	#AI_2(i_iRawSignal := 27648,
	      io_stConfig := "DB_Test_IO".Config[2],
	      io_stOut := "DB_Test_IO".Out[2]);
	#Alarm_2(i_rValue := "DB_Test_IO".Out[2].Value_Filtered, i_boReset := "DB_Test_IO".Reset_Alarms, i_boInhibit := False, io_stConfig := "DB_Test_IO".Alarm_Cfg[2], io_stOut := "DB_Test_IO".Alarm_Out[2]);
	
END_FUNCTION_BLOCK

FUNCTION_BLOCK "FB_Sim_SawTooth_UpDown"
{ S7_Optimized_Access := 'FALSE' }
VERSION : 0.1
   VAR_INPUT 
      Enable : Bool;
      Speed : Real;
      Limit_High : Int := 27648;   // Верхний предел (по умолчанию максимум для аналогового входа Siemens)
      Limit_Low : Int := 0;   // Нижний предел
   END_VAR

   VAR_OUTPUT 
      Out_Raw : Int;
   END_VAR

   VAR_IN_OUT 
      Current_Val : Int;
   END_VAR

   VAR 
      Dir_Up : Bool := TRUE;   // Направление: TRUE = вверх, FALSE = вниз
   END_VAR

   VAR_TEMP 
      Increment : Int;
   END_VAR


BEGIN
	    // Если блок выключен, замораживаем текущее значение, сохраняем направление и выходим
	    IF NOT #Enable THEN
	        #Out_Raw := #Current_Val;
	        RETURN;
	    END_IF;
	    
	    // Рассчитываем шаг за цикл
	    #Increment := REAL_TO_INT(ABS(#Speed) * "getCycleTime"() / 1000.0);
	    
	    // Логика треугольного сигнала ("вверх-вниз")
	    IF #Dir_Up THEN
	        // Считаем вверх
	        #Current_Val := #Current_Val + #Increment;
	        IF #Current_Val >= #Limit_High THEN
	            #Current_Val := #Limit_High;
	            #Dir_Up := FALSE; // Меняем направление на "вниз"
	        END_IF;
	    ELSE
	        // Считаем вниз
	        #Current_Val := #Current_Val - #Increment;
	        IF #Current_Val <= #Limit_Low THEN
	            #Current_Val := #Limit_Low;
	            #Dir_Up := TRUE;  // Меняем направление на "вверх"
	        END_IF;
	    END_IF;
	    
	    // Обновляем выход
	    #Out_Raw := #Current_Val;
	    
END_FUNCTION_BLOCK

FUNCTION "getCycleTime" : Real
{ S7_Optimized_Access := 'FALSE' }
VERSION : 0.1

BEGIN
	#getCycleTime := "DB_Global".Sys.CycleTime_ms_REAL;
END_FUNCTION

FUNCTION_BLOCK "FB_RawDistort"
{ S7_Optimized_Access := 'FALSE' }
VERSION : 0.1
// 5. BLOCKS (FB_RawDistort, FB_Sim_SawTooth, FB_AI, FB_AnalogAlarm)
   VAR_INPUT 
      Enable : Bool;
      RawIn : Int;
      Dt_ms : Real;
      NoiseAmpRaw : Int;
      Noise_Hz : Real;
      StepTrig : Bool;
      StepRaw : Int;
      StepHold_ms : DInt;
   END_VAR

   VAR_OUTPUT 
      RawOut : Int;
   END_VAR

   VAR 
      phase : Real;
      noiseVal : Real;
      step_active : Bool;
      step_left_ms : DInt;
      step_prev : Bool;
   END_VAR


BEGIN
	
	IF NOT #Enable THEN
	    #RawOut := #RawIn;
	    RETURN;
	END_IF;
	#phase := #phase + (6.283185 * #Noise_Hz * #Dt_ms * 0.001);
	IF #phase > 6.283185 THEN
	    #phase := #phase - 6.283185;
	END_IF;
	#noiseVal := SIN(#phase);
	IF (#StepTrig AND NOT #step_prev) THEN
	    #step_active := TRUE;
	    #step_left_ms := #StepHold_ms;
	END_IF;
	#step_prev := #StepTrig;
	IF #step_active THEN
	    IF #step_left_ms > REAL_TO_DINT(#Dt_ms) THEN
	        #step_left_ms := #step_left_ms - REAL_TO_DINT(#Dt_ms);
	    ELSE
	        #step_active := FALSE;
	    END_IF;
	END_IF;
	#RawOut := REAL_TO_INT(INT_TO_REAL(#RawIn) + (#noiseVal * INT_TO_REAL(#NoiseAmpRaw)));
	
END_FUNCTION_BLOCK

FUNCTION_BLOCK "FB_AI"
{ S7_Optimized_Access := 'FALSE' }
VERSION : 7.9
// -----------------------------------------------------------------------------
// БЛОК ОБРАБОТКИ АНАЛОГОВОГО СИГНАЛА (FB_AI)
// -----------------------------------------------------------------------------
   VAR_INPUT 
      i_iRawSignal : Int;
      i_rSimValue : Real;
   END_VAR

   VAR_IN_OUT 
      io_stConfig : "UDT_AI_Config";
      io_stOut : "UDT_AI_Out";
   END_VAR

   VAR 
      stat_boWasInvalid : Bool := TRUE;
   END_VAR

   VAR_TEMP 
      temp_boDisabled : Bool;
      temp_boSimActive : Bool;
      temp_boUseSqrt : Bool;
      temp_boPreSqrtCut : Bool;
      temp_boFinalClamp : Bool;
      temp_rMA : Real;
      temp_rNorm : Real;
      temp_rCutoff_Norm : Real;
      temp_rScaled : Real;
      temp_rRange_mA : Real;
      temp_rRange_Phys : Real;
      temp_rMinPhys : Real;
      temp_rMaxPhys : Real;
      temp_boResetFilter : Bool;
      temp_iFilterTime : Int;
   END_VAR


BEGIN
	    // =========================================================
	    // ШАГ 0. РАСШИФРОВКА БИТОВОГО СЛОВА (Mode)
	    // =========================================================
	    #temp_boDisabled := (#io_stConfig.Mode AND 16#0001) = 16#0001;
	    #temp_boSimActive := (#io_stConfig.Mode AND 16#0002) = 16#0002;
	    #temp_boUseSqrt := (#io_stConfig.Mode AND 16#0004) = 16#0004;
	    #temp_boPreSqrtCut := (#io_stConfig.Mode AND 16#0008) = 16#0008;
	    #temp_boFinalClamp := (#io_stConfig.Mode AND 16#0010) = 16#0010;
	    
	    // 0.1 Режим полного отключения канала
	    IF #temp_boDisabled THEN
	        #io_stOut.Value_Unclamped := 0.0;
	        #io_stOut.Value_Scaled := 0.0;
	        #io_stOut.Value_Filtered := 0.0;
	        #io_stOut.Value_mA := 0.0;
	        #io_stOut.Raw := 0;
	        
	        #io_stOut.Status.WireBreak := FALSE;
	        #io_stOut.Status.Underrange := FALSE;
	        #io_stOut.Status.Overrange := FALSE;
	        #io_stOut.Status.Overflow := FALSE;
	        #io_stOut.Status.ConfigError := FALSE;
	        #io_stOut.Status.Sim_Active := FALSE;
	        
	        #stat_boWasInvalid := TRUE;
	        RETURN;
	    END_IF;
	    
	    // 0.2 Защита от кривых настроек
	    #temp_rRange_mA := #io_stConfig.Calib_mA_Max - #io_stConfig.Calib_mA_Min;
	    #temp_rRange_Phys := #io_stConfig.Scale_Max - #io_stConfig.Scale_Min;
	    
	    IF (#io_stConfig.HW_Max <= #io_stConfig.HW_Min) OR
	        (#temp_rRange_mA <= 0.0) OR
	        (ABS(#temp_rRange_Phys) < 0.00001) OR
	        (ABS(#io_stConfig.Cutoff) >= ABS(#temp_rRange_Phys)) THEN
	        
	        #io_stOut.Status.ConfigError := TRUE;
	        
	        #io_stOut.Status.WireBreak := FALSE;
	        #io_stOut.Status.Underrange := FALSE;
	        #io_stOut.Status.Overrange := FALSE;
	        #io_stOut.Status.Overflow := FALSE;
	        #io_stOut.Status.Sim_Active := FALSE;
	        
	        #io_stOut.Value_Unclamped := 0.0;
	        #io_stOut.Value_Scaled := 0.0;
	        #io_stOut.Value_Filtered := 0.0;
	        #io_stOut.Value_mA := 0.0;
	        #io_stOut.Raw := #i_iRawSignal;
	        
	        #stat_boWasInvalid := TRUE;
	        RETURN;
	    END_IF;
	    
	    #io_stOut.Status.ConfigError := FALSE;
	    
	    // =========================================================
	    // ШАГ 1 & 2. СИМУЛЯЦИЯ И ДИАГНОСТИКА
	    // =========================================================
	    
	    IF #temp_boSimActive THEN
	        #io_stOut.Status.Sim_Active := TRUE;
	        
	        #io_stOut.Status.WireBreak := FALSE;
	        #io_stOut.Status.Underrange := FALSE;
	        #io_stOut.Status.Overrange := FALSE;
	        #io_stOut.Status.Overflow := FALSE;
	        
	        #io_stOut.Raw := 0;
	        #io_stOut.Value_mA := 0.0;
	        #temp_rScaled := #i_rSimValue;
	    ELSE
	        #io_stOut.Status.Sim_Active := FALSE;
	        #io_stOut.Raw := #i_iRawSignal;
	        
	        "FC_AnalogDiag"(
	                        i_iRawSignal := #i_iRawSignal,
	                        i_iHW_Min := #io_stConfig.HW_Min,
	                        i_iHW_Max := #io_stConfig.HW_Max,
	                        i_rCoef_Under := "C_DIAG_UNDER",
	                        i_rCoef_Over := "C_DIAG_OVER",
	                        o_boWireBreak => #io_stOut.Status.WireBreak,
	                        o_boUnderrange => #io_stOut.Status.Underrange,
	                        o_boOverrange => #io_stOut.Status.Overrange,
	                        o_boOverflow => #io_stOut.Status.Overflow
	        );
	        
	        // =========================================================
	        // ШАГ 3. МАТЕМАТИКА
	        // =========================================================
	        IF #io_stOut.Status.WireBreak THEN
	            // Ушли в жесткий минус: База + (Диапазон * Коэффициент обрыва)
	            #temp_rScaled := #io_stConfig.Scale_Min + (#temp_rRange_Phys * "C_DIAG_UNDER");
	            #io_stOut.Value_mA := 0.0;
	            
	        ELSIF #io_stOut.Status.Overflow THEN
	            // Ушли в жесткий перегруз: База + (Диапазон * Коэффициент переполнения)
	            #temp_rScaled := #io_stConfig.Scale_Min + (#temp_rRange_Phys * "C_DIAG_OVER");
	            #io_stOut.Value_mA := 25.0;
	        ELSE
	            // А) Расчет миллиампер
	            #temp_rMA := 4.0 + ((INT_TO_REAL(#i_iRawSignal) - INT_TO_REAL(#io_stConfig.HW_Min)) /
	            (INT_TO_REAL(#io_stConfig.HW_Max) - INT_TO_REAL(#io_stConfig.HW_Min))) * 16.0;
	            #io_stOut.Value_mA := #temp_rMA;
	            
	            // Б) Нормализация (0.0 ... 1.0)
	            #temp_rNorm := (#temp_rMA - #io_stConfig.Calib_mA_Min) / #temp_rRange_mA;
	            
	            // В) Pre-Sqrt CutOff (Умная отсечка до извлечения корня)
	            IF #temp_boPreSqrtCut AND #temp_boUseSqrt THEN
	                #temp_rCutoff_Norm := ABS(#io_stConfig.Cutoff / #temp_rRange_Phys);
	                #temp_rCutoff_Norm := #temp_rCutoff_Norm * #temp_rCutoff_Norm;
	                
	                IF #temp_rNorm < #temp_rCutoff_Norm THEN
	                    #temp_rNorm := 0.0;
	                END_IF;
	            END_IF;
	            
	            // Г) Извлечение корня
	            IF #temp_boUseSqrt THEN
	                IF #temp_rNorm > 0.0 THEN
	                    #temp_rNorm := SQRT(#temp_rNorm);
	                ELSE
	                    #temp_rNorm := 0.0;
	                END_IF;
	            END_IF;
	            
	            // Д) Масштабирование в физическую величину
	            #temp_rScaled := #io_stConfig.Scale_Min + (#temp_rNorm * #temp_rRange_Phys);
	            
	            // Е) Классический CutOff 
	            IF NOT (#temp_boPreSqrtCut AND #temp_boUseSqrt) THEN
	                IF ABS(#temp_rScaled) < ABS(#io_stConfig.Cutoff) THEN
	                    #temp_rScaled := 0.0;
	                END_IF;
	            END_IF;
	        END_IF;
	    END_IF;
	    
	    // Сохраняем чистую математику (без клампа) на выход
	    #io_stOut.Value_Unclamped := #temp_rScaled;
	    
	    // =========================================================
	    // ШАГ 3.5. ФИНАЛЬНЫЙ CLAMP (Beautiful Branch)
	    // =========================================================
	    IF #temp_boFinalClamp THEN
	        #temp_rMinPhys := MIN(IN1 := #io_stConfig.Scale_Min, IN2 := #io_stConfig.Scale_Max);
	        #temp_rMaxPhys := MAX(IN1 := #io_stConfig.Scale_Min, IN2 := #io_stConfig.Scale_Max);
	        #temp_rScaled := LIMIT(MN := #temp_rMinPhys, IN := #temp_rScaled, MX := #temp_rMaxPhys);
	    END_IF;
	    
	    #io_stOut.Value_Scaled := #temp_rScaled;
	    
	    // =========================================================
	    // ШАГ 4. ФИЛЬТРАЦИЯ & PRE-LOAD 
	    // =========================================================
	    #temp_boResetFilter := #temp_boSimActive OR
	    #io_stOut.Status.WireBreak OR
	    #io_stOut.Status.Overflow OR
	    #stat_boWasInvalid;
	    
	    #temp_iFilterTime := LIMIT(MN := 0, IN := #io_stConfig.FilterTime_ms, MX := 32000);
	    
	    "FC_Filter_PT1"(
	                    i_rRawValue := #temp_rScaled, // Фильтруем заклампованное значение
	                    i_rTimeFilter_ms := INT_TO_REAL(#temp_iFilterTime),
	                    i_boReset := #temp_boResetFilter,
	                    io_rFilteredValue := #io_stOut.Value_Filtered
	    );
	    
	    #stat_boWasInvalid := #io_stOut.Status.WireBreak OR
	    #io_stOut.Status.Overflow OR
	    #io_stOut.Status.ConfigError;
	    
END_FUNCTION_BLOCK

FUNCTION "FC_AnalogDiag" : Void
{ S7_Optimized_Access := 'FALSE' }
VERSION : 1.1
   VAR_INPUT 
      i_iRawSignal : Int;
      i_iHW_Min : Int;
      i_iHW_Max : Int;
      i_rCoef_Under : Real;
      i_rCoef_Over : Real;
   END_VAR

   VAR_OUTPUT 
      o_boWireBreak : Bool;
      o_boUnderrange : Bool;
      o_boOverrange : Bool;
      o_boOverflow : Bool;
   END_VAR

   VAR_TEMP 
      temp_rLimit_Max : Real;
      temp_iLimit_Min : Int;
   END_VAR


BEGIN
	    #temp_rLimit_Max := INT_TO_REAL(#i_iHW_Max) * #i_rCoef_Over;
	    #temp_iLimit_Min := REAL_TO_INT(INT_TO_REAL(#i_iHW_Max) * #i_rCoef_Under);
	    
	    #o_boWireBreak := #i_iRawSignal < #temp_iLimit_Min;
	    #o_boUnderrange := (#i_iRawSignal < #i_iHW_Min) AND (#i_iRawSignal >= #temp_iLimit_Min);
	    #o_boOverrange := (#i_iRawSignal > #i_iHW_Max) AND (#i_iRawSignal <= REAL_TO_INT(#temp_rLimit_Max));
	    #o_boOverflow := #i_iRawSignal > REAL_TO_INT(#temp_rLimit_Max);
END_FUNCTION

FUNCTION "FC_Filter_PT1" : Void
{ S7_Optimized_Access := 'FALSE' }
VERSION : 0.1
   VAR_INPUT 
      i_rRawValue : Real;
      i_rTimeFilter_ms : Real;
      i_boReset : Bool;
   END_VAR

   VAR_IN_OUT 
      io_rFilteredValue : Real;
   END_VAR

   VAR_TEMP 
      temp_rCycleTime_ms : Real;
      temp_rAlpha : Real;
   END_VAR


BEGIN
	
	IF #i_boReset THEN
	    #io_rFilteredValue := #i_rRawValue;
	    RETURN;
	END_IF;
	#temp_rCycleTime_ms := "getCycleTime"();
	IF #temp_rCycleTime_ms <= 0.000001 THEN
	    RETURN;
	END_IF;
	#temp_rAlpha := #temp_rCycleTime_ms / (#i_rTimeFilter_ms + #temp_rCycleTime_ms);
	#io_rFilteredValue := #io_rFilteredValue + #temp_rAlpha * (#i_rRawValue - #io_rFilteredValue);
	
	
	
END_FUNCTION

FUNCTION_BLOCK "FB_AnalogAlarm"
{ S7_Optimized_Access := 'FALSE' }
VERSION : 2.0
   VAR_INPUT 
      i_rValue : Real;
      i_boReset : Bool;
      i_boInhibit : Bool;
   END_VAR

   VAR_IN_OUT 
      io_stConfig : "UDT_Alarm_Config";
      io_stOut : "UDT_Alarm_Out";
   END_VAR

   VAR 
      stat_TonHiHi {InstructionName := 'TON'; LibVersion := '1.0'; S7_SetPoint := 'False'} : TON;
      stat_TonHi {InstructionName := 'TON'; LibVersion := '1.0'; S7_SetPoint := 'False'} : TON;
      stat_TonLo {InstructionName := 'TON'; LibVersion := '1.0'; S7_SetPoint := 'False'} : TON;
      stat_TonLoLo {InstructionName := 'TON'; LibVersion := '1.0'; S7_SetPoint := 'False'} : TON;
      stat_RawHiHi : Bool;
      stat_RawHi : Bool;
      stat_RawLo : Bool;
      stat_RawLoLo : Bool;
   END_VAR


BEGIN
	    // =========================================================
	    // 1. ТРАНСЛЯЦИЯ СТАТУСОВ ДЛЯ HMI (En_Out)
	    // =========================================================
	    #io_stOut.En_HiHi := #io_stConfig.En_Alarm.HiHi AND NOT #i_boInhibit ;
	    #io_stOut.En_Hi := #io_stConfig.En_Alarm.Hi AND NOT #i_boInhibit;
	    #io_stOut.En_Lo := #io_stConfig.En_Alarm.Lo AND NOT #i_boInhibit;
	    #io_stOut.En_LoLo := #io_stConfig.En_Alarm.LoLo AND NOT #i_boInhibit;
	    #io_stOut.En_Latch_Enable := #io_stConfig.En_Alarm.Latch_Enable;
	    
	    // =========================================================
	    // 2. ОБРАБОТКА СЫРЫХ АВАРИЙ С ГИСТЕРЕЗИСОМ (Deadband)
	    // =========================================================
	    // Верхние пороги (Срабатывание >, Сброс <)
	    IF #i_rValue > #io_stConfig.HiHi THEN
	        #stat_RawHiHi := TRUE;
	    ELSIF #i_rValue < (#io_stConfig.HiHi - #io_stConfig.Hysteresis) THEN
	        #stat_RawHiHi := FALSE;
	    END_IF;
	    
	    IF #i_rValue > #io_stConfig.Hi THEN
	        #stat_RawHi := TRUE;
	    ELSIF #i_rValue < (#io_stConfig.Hi - #io_stConfig.Hysteresis) THEN
	        #stat_RawHi := FALSE;
	    END_IF;
	    
	    // Нижние пороги (Срабатывание <, Сброс >)
	    IF #i_rValue < #io_stConfig.Lo THEN
	        #stat_RawLo := TRUE;
	    ELSIF #i_rValue > (#io_stConfig.Lo + #io_stConfig.Hysteresis) THEN
	        #stat_RawLo := FALSE;
	    END_IF;
	    
	    IF #i_rValue < #io_stConfig.LoLo THEN
	        #stat_RawLoLo := TRUE;
	    ELSIF #i_rValue > (#io_stConfig.LoLo + #io_stConfig.Hysteresis) THEN
	        #stat_RawLoLo := FALSE;
	    END_IF;
	    
	    // =========================================================
	    // 3. ТАЙМЕРЫ ЗАДЕРЖКИ (ON-Delay)
	    // =========================================================
	    // Таймер не считает, если сработала блокировка датчика (Inhibit) 
	    // или аларм выключен в настройках.
	    #stat_TonHiHi(IN := #stat_RawHiHi AND #io_stConfig.En_Alarm.HiHi AND NOT #i_boInhibit,
	                  PT := DINT_TO_TIME(#io_stConfig.Delay_HiHi)*1000 );
	    
	    #stat_TonHi(IN := #stat_RawHi AND #io_stConfig.En_Alarm.Hi AND NOT #i_boInhibit,
	                PT := DINT_TO_TIME(#io_stConfig.Delay_Hi)*1000 );
	    
	    #stat_TonLo(IN := #stat_RawLo AND #io_stConfig.En_Alarm.Lo AND NOT #i_boInhibit,
	                PT := DINT_TO_TIME(#io_stConfig.Delay_Lo)*1000 );
	    
	    #stat_TonLoLo(IN := #stat_RawLoLo AND #io_stConfig.En_Alarm.LoLo AND NOT #i_boInhibit,
	                  PT := DINT_TO_TIME(#io_stConfig.Delay_LoLo)*1000 );
	    
	    // =========================================================
	    // 4. ФИКСАЦИЯ (LATCH) И СБРОС АВАРИЙ
	    // =========================================================
	    // Логика сброса (имеет приоритет):
	    // 1. Сработал Inhibit (глушим всё безусловно)
	    // 2. Аларм сняли в настройках
	    // 3. Уровень в норме И (нет фиксации ИЛИ нажата кнопка Reset)
	    
	    // --- HiHi ---
	    IF #i_boInhibit OR NOT #io_stConfig.En_Alarm.HiHi OR
	        (NOT #stat_RawHiHi AND (NOT #io_stConfig.En_Alarm.Latch_Enable OR #i_boReset)) THEN
	        #io_stOut.HiHi := FALSE;
	    ELSIF #stat_TonHiHi.Q THEN
	        #io_stOut.HiHi := TRUE;
	    END_IF;
	    
	    // --- Hi ---
	    IF #i_boInhibit OR NOT #io_stConfig.En_Alarm.Hi OR
	        (NOT #stat_RawHi AND (NOT #io_stConfig.En_Alarm.Latch_Enable OR #i_boReset)) THEN
	        #io_stOut.Hi := FALSE;
	    ELSIF #stat_TonHi.Q THEN
	        #io_stOut.Hi := TRUE;
	    END_IF;
	    
	    // --- Lo ---
	    IF #i_boInhibit OR NOT #io_stConfig.En_Alarm.Lo OR
	        (NOT #stat_RawLo AND (NOT #io_stConfig.En_Alarm.Latch_Enable OR #i_boReset)) THEN
	        #io_stOut.Lo := FALSE;
	    ELSIF #stat_TonLo.Q THEN
	        #io_stOut.Lo := TRUE;
	    END_IF;
	    
	    // --- LoLo ---
	    IF #i_boInhibit OR NOT #io_stConfig.En_Alarm.LoLo OR
	        (NOT #stat_RawLoLo AND (NOT #io_stConfig.En_Alarm.Latch_Enable OR #i_boReset)) THEN
	        #io_stOut.LoLo := FALSE;
	    ELSIF #stat_TonLoLo.Q THEN
	        #io_stOut.LoLo := TRUE;
	    END_IF;
	    
END_FUNCTION_BLOCK

FUNCTION "FC_Wh_TRN_Mng" : Void
{ S7_Optimized_Access := 'FALSE' }
VERSION : 0.1
   VAR_TEMP 
      temp_Ind : Int;
   END_VAR


BEGIN
	// ---------------------------------------------------------------
	// Склад: Транзитный (TRN) — 2 весовых и 1 аналоговый
	// ---------------------------------------------------------------
	
	"iDB_TRN_Tank_Log_1"(i_iRaw_AI := "DB_IO_MAP".AI_TRN_Tank_1,
	                     i_rRaw_Siwa := 0.0,
	                     i_boRaw_DI := "DB_IO_MAP".DI_TRN_Tank_1,
	                     io_Tank := "DB_Wh_TRN".Tank[1]);
	
	
	"iDB_TRN_Tank_Log_2"(i_iRaw_AI := 0,
	                     i_rRaw_Siwa := "DB_IO_MAP".AI_TRN_WTank_2,
	                     i_boRaw_DI := "DB_IO_MAP".DI_TRN_WTank_2,
	                     io_Tank := "DB_Wh_TRN".Tank[2]);
	
	"iDB_TRN_Tank_Log_3"(i_iRaw_AI := 0,
	                     i_rRaw_Siwa := "DB_IO_MAP".AI_TRN_WTank_3,
	                     i_boRaw_DI := "DB_IO_MAP".DI_TRN_WTank_3,
	                     io_Tank := "DB_Wh_TRN".Tank[3]);
	
	FOR #temp_Ind := 1 TO "c_Count_TRN" DO
	    "FC_Map_SmallTank_HMI"(io_Tank_Internal := "DB_Wh_TRN".Tank[#temp_Ind],
	                           io_HMI_Tank := "DB_HMI_MAP".TRN_SmalTank[#temp_Ind]);
	END_FOR;
	
END_FUNCTION

FUNCTION "FC_Map_SmallTank_HMI" : Void
TITLE = Маппинг HMI малого танка
{ S7_Optimized_Access := 'FALSE' }
AUTHOR : S7A_Lib
FAMILY : HMI_Map
VERSION : 0.2
// ==============================================================================
// Описание: Перекладывает данные из внутренней структуры малого танка 
//           в плоскую HMI-структуру. Включает конвертацию массы в тонны 
//           и сквозную передачу статусных битов.
// ==============================================================================
   VAR_IN_OUT 
      io_Tank_Internal : "UDT_Tank_Full";   // Рабочая (внутренняя) структура танка
      io_HMI_Tank : "UDT_HMI_SmallTank";   // Плоская структура для панели оператора
   END_VAR


BEGIN
	        // --- Основные технологические параметры ---
	        #io_HMI_Tank.Level_m := #io_Tank_Internal.Calc.Level_m;
	        #io_HMI_Tank.Volume_m3 := #io_Tank_Internal.Calc.Volume_m3;
	        #io_HMI_Tank.Level_pct := #io_Tank_Internal.Calc.Level_Pct;
	        #io_HMI_Tank.Weight_t := #io_Tank_Internal.Calc.Weight_t;
	        
	        // --- Минимально фильтруем убрав шубу ---
	        "FC_Filter_PT1"(i_rRawValue := #io_Tank_Internal.AI_Out.Value_Unclamped,
	                        i_rTimeFilter_ms := 100.0,
	                        i_boReset := "isFirstScan"(),
	                        io_rFilteredValue := #io_HMI_Tank.Level_Raw_m);
	        
	        // --- Геометрия для шкалы HMI ---
	        #io_HMI_Tank.Height_Full_m := #io_Tank_Internal.Geom.Height_Full_m;
	        
	        // --- Статусные биты аварий ---
	        #io_HMI_Tank.Alarm_DI := #io_Tank_Internal.DI_Alarm.Alarm;
	        #io_HMI_Tank.Alarm_HH := #io_Tank_Internal.AI_Alarm.HiHi;
	        #io_HMI_Tank.Alarm_H := #io_Tank_Internal.AI_Alarm.Hi;
	        #io_HMI_Tank.Alarm_L := #io_Tank_Internal.AI_Alarm.Lo;
	        #io_HMI_Tank.Alarm_LL := #io_Tank_Internal.AI_Alarm.LoLo;
	        
	        #io_HMI_Tank.Status_DI_Disabled := #io_Tank_Internal.DI_Out.Disabled;
	        #io_HMI_Tank.Status_DI_Value := #io_Tank_Internal.DI_Out.Value;
	        // --- Диагностика AI ---
	        #io_HMI_Tank.Status_AI_Disabled := #io_Tank_Internal.AI_Out.Status.Disabled;
	        #io_HMI_Tank.Status_AI_WireBreak := #io_Tank_Internal.AI_Out.Status.WireBreak;
	        #io_HMI_Tank.Status_AI_Underrange := #io_Tank_Internal.AI_Out.Status.Underrange;
	        #io_HMI_Tank.Status_AI_Overrange := #io_Tank_Internal.AI_Out.Status.Overrange;
	        #io_HMI_Tank.Status_AI_Overflow := #io_Tank_Internal.AI_Out.Status.Overflow;
	        #io_HMI_Tank.Status_AI_ConfigError := #io_Tank_Internal.AI_Out.Status.ConfigError;
	        
	        // --- Команды HMI -> Tank (сброс ошибок) ---
	        #io_Tank_Internal.Cmd.ResetError := #io_HMI_Tank.Cmd_Reset;
	        #io_HMI_Tank.Cmd_Reset := FALSE;
	        
END_FUNCTION

FUNCTION "isFirstScan" : Bool
{ S7_Optimized_Access := 'FALSE' }
VERSION : 0.1

BEGIN
	#isFirstScan := "DB_Global".Sys.FirstScan;
END_FUNCTION

FUNCTION "FC_Scale_Map_Mng" : Void
{ S7_Optimized_Access := 'FALSE' }
VERSION : 0.1

BEGIN
	"iDB_Map_Siwarex_Core_1"(i_Scale_DB:="DB_Scale_CS_1",
	                         i_CycleTime_ms:=0,
	                         io_Core:="DB_MAP".Scale_CS_1);
	
	"iDB_Map_Siwarex_Core_2"(i_Scale_DB:="DB_Scale_CS_2",
	                         i_CycleTime_ms:=0,
	                         io_Core:="DB_MAP".Scale_CS_2);
	
END_FUNCTION

FUNCTION "FC_Wh_POL_Mng" : Void
{ S7_Optimized_Access := 'FALSE' }
VERSION : 0.1

BEGIN
	"iDB_POL_Tank_Log_1"(i_iRaw_AI:="DB_IO_MAP".AI_POL_Tank_1,
	                 i_rRaw_Siwa:=0.0,
	                 i_boRaw_DI:="DB_IO_MAP".DI_POL_Tank_1,
	                 io_Tank:="DB_Wh_POL".Tank[1]);
	
	"iDB_POL_Tank_Log_2"(i_iRaw_AI := "DB_IO_MAP".AI_POL_Tank_2,
	                     i_rRaw_Siwa := 0.0,
	                     i_boRaw_DI := "DB_IO_MAP".DI_POL_Tank_2,
	                     io_Tank := "DB_Wh_POL".Tank[2]);
	
	"iDB_POL_Tank_Log_3"(i_iRaw_AI:="DB_IO_MAP".AI_POL_Tank_3,
	                     i_rRaw_Siwa:=0.0,
	                     i_boRaw_DI:="DB_IO_MAP".DI_POL_Tank_3,
	                     io_Tank:="DB_Wh_POL".Tank[3]);
	
END_FUNCTION

ORGANIZATION_BLOCK "OB121"   // OB121, FBD, ProgrammingError
VERSION : 0.1
// stored: IsIECCheckEnabled false
   VAR_TEMP
      Temp_0 : Byte;
      Temp_1 : Byte;
      Temp_2 : Byte;
      Temp_3 : Byte;
      Temp_4 : Byte;
      Temp_5 : Byte;
      Temp_6 : Word;
      Temp_7 : Word;
      Temp_8 : Word;
      Temp_9 : Date_And_Time;
   END_VAR
BEGIN
END_ORGANIZATION_BLOCK

ORGANIZATION_BLOCK "OB122"   // OB122, FBD, IOAccessError
VERSION : 0.1
// stored: IsIECCheckEnabled false
   VAR_TEMP
      Temp_0 : Byte;
      Temp_1 : Byte;
      Temp_2 : Byte;
      Temp_3 : Byte;
      Temp_4 : Byte;
      Temp_5 : Byte;
      Temp_6 : Word;
      Temp_7 : Word;
      Temp_8 : Word;
      Temp_9 : Date_And_Time;
   END_VAR
BEGIN
END_ORGANIZATION_BLOCK

ORGANIZATION_BLOCK "OB80"   // OB80, FBD, TimeErrorInterrupt
VERSION : 0.1
// stored: IsIECCheckEnabled false
   VAR_TEMP
      Temp_0 : Byte;
      Temp_1 : Byte;
      Temp_2 : Byte;
      Temp_3 : Byte;
      Temp_4 : Byte;
      Temp_5 : Byte;
      Temp_6 : Word;
      Temp_7 : Byte;
      Temp_8 : Byte;
      Temp_9 : Byte;
      Temp_10 : Byte;
      Temp_11 : Date_And_Time;
   END_VAR
BEGIN
END_ORGANIZATION_BLOCK

ORGANIZATION_BLOCK "OB82"   // OB82, FBD, DiagnosticErrorInterrupt
VERSION : 0.1
// stored: IsIECCheckEnabled false
   VAR_TEMP
      Temp_0 : Byte;
      Temp_1 : Byte;
      Temp_2 : Byte;
      Temp_3 : Byte;
      Temp_4 : Byte;
      Temp_5 : Byte;
      Temp_6 : Word;
      Temp_7 : Bool;
      Temp_8 : Bool;
      Temp_9 : Bool;
      Temp_10 : Bool;
      Temp_11 : Bool;
      Temp_12 : Bool;
      Temp_13 : Bool;
      Temp_14 : Bool;
      Temp_15 : Byte;
      Temp_16 : Bool;
      Temp_17 : Bool;
      Temp_18 : Bool;
      Temp_19 : Bool;
      Temp_20 : Bool;
      Temp_21 : Bool;
      Temp_22 : Bool;
      Temp_23 : Bool;
      Temp_24 : Bool;
      Temp_25 : Bool;
      Temp_26 : Bool;
      Temp_27 : Bool;
      Temp_28 : Bool;
      Temp_29 : Bool;
      Temp_30 : Bool;
      Temp_31 : Bool;
      Temp_32 : Date_And_Time;
   END_VAR
BEGIN
END_ORGANIZATION_BLOCK

ORGANIZATION_BLOCK "OB83"   // OB83, FBD, PullOrPlugOfModules
VERSION : 0.1
// stored: IsIECCheckEnabled false
   VAR_TEMP
      Temp_0 : Byte;
      Temp_1 : Byte;
      Temp_2 : Byte;
      Temp_3 : Byte;
      Temp_4 : Byte;
      Temp_5 : Byte;
      Temp_6 : Word;
      Temp_7 : Int;
      Temp_8 : Word;
      Temp_9 : Date_And_Time;
   END_VAR
BEGIN
END_ORGANIZATION_BLOCK

ORGANIZATION_BLOCK "OB85"   // OB85, FBD, AccessError
VERSION : 0.1
// stored: IsIECCheckEnabled false
   VAR_TEMP
      Temp_0 : Byte;
      Temp_1 : Byte;
      Temp_2 : Byte;
      Temp_3 : Byte;
      Temp_4 : Byte;
      Temp_5 : Byte;
      Temp_6 : Int;
      Temp_7 : Byte;
      Temp_8 : Byte;
      Temp_9 : Byte;
      Temp_10 : Byte;
      Temp_11 : Date_And_Time;
   END_VAR
BEGIN
END_ORGANIZATION_BLOCK

ORGANIZATION_BLOCK "OB86"   // OB86, FBD, RackOrStationFailure
VERSION : 0.1
// stored: IsIECCheckEnabled false
   VAR_TEMP
      Temp_0 : Byte;
      Temp_1 : Byte;
      Temp_2 : Byte;
      Temp_3 : Byte;
      Temp_4 : Byte;
      Temp_5 : Byte;
      Temp_6 : Word;
      Temp_7 : Array[0..31] of Bool;
      Temp_8 : Date_And_Time;
   END_VAR
BEGIN
END_ORGANIZATION_BLOCK

ORGANIZATION_BLOCK "OB87"   // OB87, FBD, CommunicationError
VERSION : 0.1
// stored: IsIECCheckEnabled false
   VAR_TEMP
      Temp_0 : Byte;
      Temp_1 : Byte;
      Temp_2 : Byte;
      Temp_3 : Byte;
      Temp_4 : Byte;
      Temp_5 : Byte;
      Temp_6 : Word;
      Temp_7 : DWord;
      Temp_8 : Date_And_Time;
   END_VAR
BEGIN
END_ORGANIZATION_BLOCK

FUNCTION "FC_Scale_Instance" : Void   // FC19, FBD
VERSION : 0.1
// stored: AutoNumber true, IsIECCheckEnabled false, UDAEnableTagReadback false
BEGIN

REGION Network 1
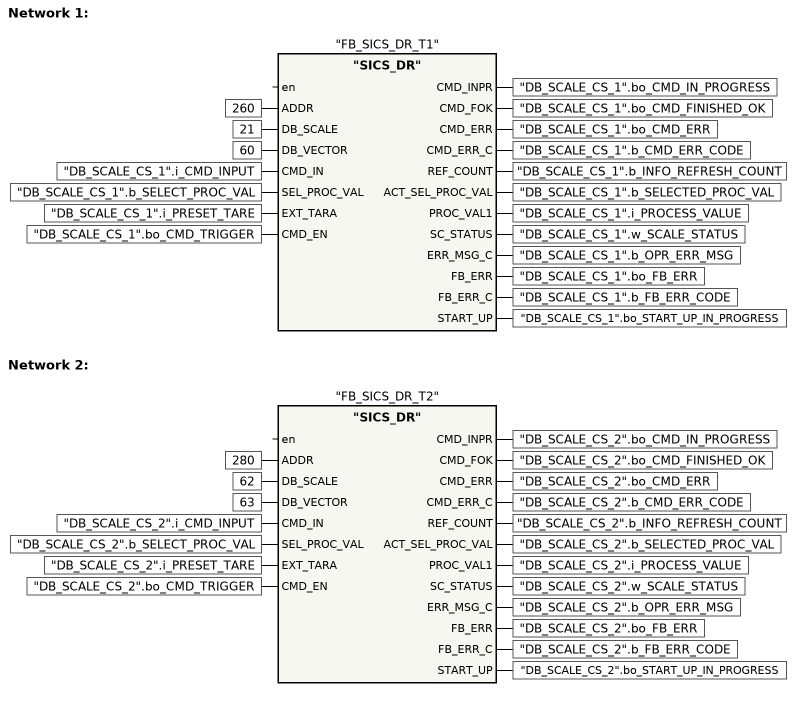
   "FB_SICS_DR_T1"(ADDR := 260,   // "SICS_DR"
                   DB_SCALE := 21,
                   DB_VECTOR := 60,
                   CMD_IN := "DB_SCALE_CS_1".i_CMD_INPUT,
                   SEL_PROC_VAL := "DB_SCALE_CS_1".b_SELECT_PROC_VAL,
                   EXT_TARA := "DB_SCALE_CS_1".i_PRESET_TARE,
                   CMD_EN := "DB_SCALE_CS_1".bo_CMD_TRIGGER,
                   CMD_INPR => "DB_SCALE_CS_1".bo_CMD_IN_PROGRESS,
                   CMD_FOK => "DB_SCALE_CS_1".bo_CMD_FINISHED_OK,
                   CMD_ERR => "DB_SCALE_CS_1".bo_CMD_ERR,
                   CMD_ERR_C => "DB_SCALE_CS_1".b_CMD_ERR_CODE,
                   REF_COUNT => "DB_SCALE_CS_1".b_INFO_REFRESH_COUNT,
                   ACT_SEL_PROC_VAL => "DB_SCALE_CS_1".b_SELECTED_PROC_VAL,
                   PROC_VAL1 => "DB_SCALE_CS_1".i_PROCESS_VALUE,
                   SC_STATUS => "DB_SCALE_CS_1".w_SCALE_STATUS,
                   ERR_MSG_C => "DB_SCALE_CS_1".b_OPR_ERR_MSG,
                   FB_ERR => "DB_SCALE_CS_1".bo_FB_ERR,
                   FB_ERR_C => "DB_SCALE_CS_1".b_FB_ERR_CODE,
                   START_UP => "DB_SCALE_CS_1".bo_START_UP_IN_PROGRESS);
END_REGION

REGION Network 2
   "FB_SICS_DR_T2"(ADDR := 280,   // "SICS_DR"
                   DB_SCALE := 62,
                   DB_VECTOR := 63,
                   CMD_IN := "DB_SCALE_CS_2".i_CMD_INPUT,
                   SEL_PROC_VAL := "DB_SCALE_CS_2".b_SELECT_PROC_VAL,
                   EXT_TARA := "DB_SCALE_CS_2".i_PRESET_TARE,
                   CMD_EN := "DB_SCALE_CS_2".bo_CMD_TRIGGER,
                   CMD_INPR => "DB_SCALE_CS_2".bo_CMD_IN_PROGRESS,
                   CMD_FOK => "DB_SCALE_CS_2".bo_CMD_FINISHED_OK,
                   CMD_ERR => "DB_SCALE_CS_2".bo_CMD_ERR,
                   CMD_ERR_C => "DB_SCALE_CS_2".b_CMD_ERR_CODE,
                   REF_COUNT => "DB_SCALE_CS_2".b_INFO_REFRESH_COUNT,
                   ACT_SEL_PROC_VAL => "DB_SCALE_CS_2".b_SELECTED_PROC_VAL,
                   PROC_VAL1 => "DB_SCALE_CS_2".i_PROCESS_VALUE,
                   SC_STATUS => "DB_SCALE_CS_2".w_SCALE_STATUS,
                   ERR_MSG_C => "DB_SCALE_CS_2".b_OPR_ERR_MSG,
                   FB_ERR => "DB_SCALE_CS_2".bo_FB_ERR,
                   FB_ERR_C => "DB_SCALE_CS_2".b_FB_ERR_CODE,
                   START_UP => "DB_SCALE_CS_2".bo_START_UP_IN_PROGRESS);
END_REGION
END_FUNCTION

FUNCTION "FC_Scale_Mng" : Void   // FC19, FBD
VERSION : 0.1
// stored: AutoNumber true, IsIECCheckEnabled false, UDAEnableTagReadback false
BEGIN

REGION Network 1
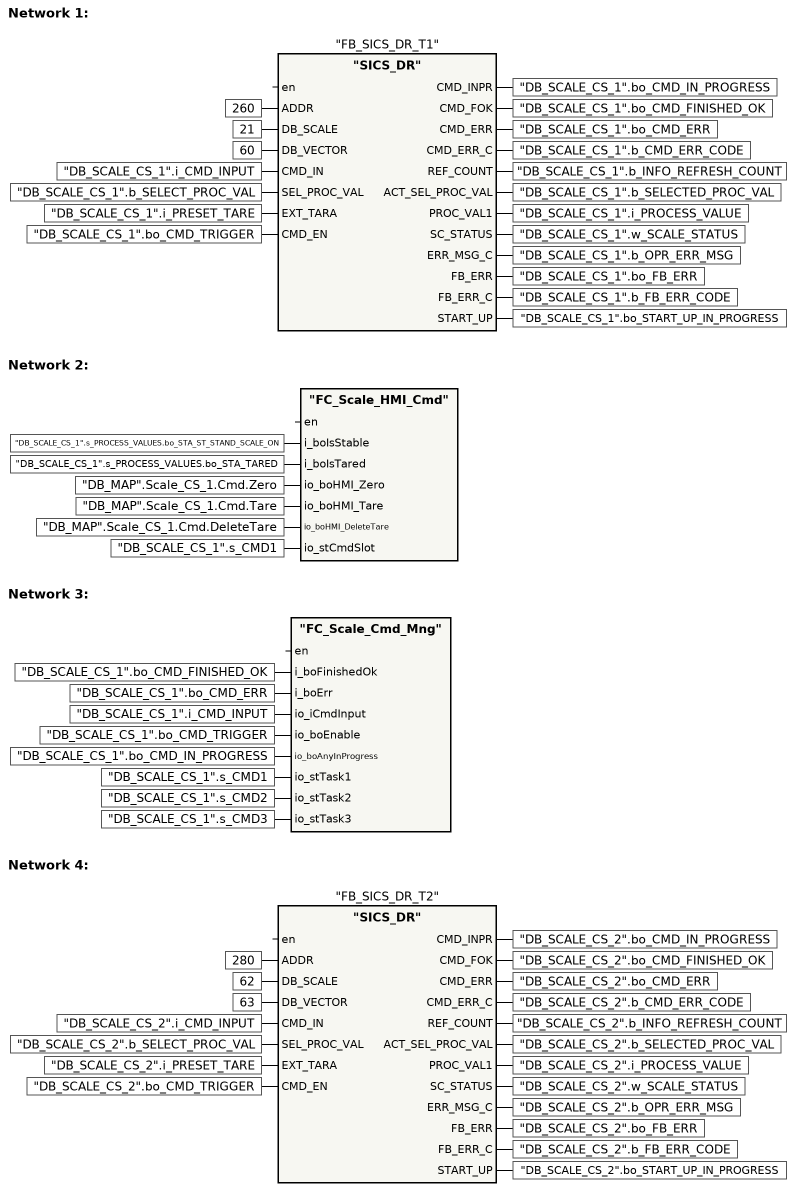
   "FB_SICS_DR_T1"(ADDR := 260,   // "SICS_DR"
                   DB_SCALE := 21,
                   DB_VECTOR := 60,
                   CMD_IN := "DB_SCALE_CS_1".i_CMD_INPUT,
                   SEL_PROC_VAL := "DB_SCALE_CS_1".b_SELECT_PROC_VAL,
                   EXT_TARA := "DB_SCALE_CS_1".i_PRESET_TARE,
                   CMD_EN := "DB_SCALE_CS_1".bo_CMD_TRIGGER,
                   CMD_INPR => "DB_SCALE_CS_1".bo_CMD_IN_PROGRESS,
                   CMD_FOK => "DB_SCALE_CS_1".bo_CMD_FINISHED_OK,
                   CMD_ERR => "DB_SCALE_CS_1".bo_CMD_ERR,
                   CMD_ERR_C => "DB_SCALE_CS_1".b_CMD_ERR_CODE,
                   REF_COUNT => "DB_SCALE_CS_1".b_INFO_REFRESH_COUNT,
                   ACT_SEL_PROC_VAL => "DB_SCALE_CS_1".b_SELECTED_PROC_VAL,
                   PROC_VAL1 => "DB_SCALE_CS_1".i_PROCESS_VALUE,
                   SC_STATUS => "DB_SCALE_CS_1".w_SCALE_STATUS,
                   ERR_MSG_C => "DB_SCALE_CS_1".b_OPR_ERR_MSG,
                   FB_ERR => "DB_SCALE_CS_1".bo_FB_ERR,
                   FB_ERR_C => "DB_SCALE_CS_1".b_FB_ERR_CODE,
                   START_UP => "DB_SCALE_CS_1".bo_START_UP_IN_PROGRESS);
END_REGION

REGION Network 2
   "FC_Scale_HMI_Cmd"(i_boIsStable := "DB_SCALE_CS_1".s_PROCESS_VALUES.bo_STA_ST_STAND_SCALE_ON,
                      i_boIsTared := "DB_SCALE_CS_1".s_PROCESS_VALUES.bo_STA_TARED,
                      io_boHMI_Zero := "DB_MAP".Scale_CS_1.Cmd.Zero,
                      io_boHMI_Tare := "DB_MAP".Scale_CS_1.Cmd.Tare,
                      io_boHMI_DeleteTare := "DB_MAP".Scale_CS_1.Cmd.DeleteTare,
                      io_stCmdSlot := "DB_SCALE_CS_1".s_CMD1);
END_REGION

REGION Network 3
   "FC_Scale_Cmd_Mng"(i_boFinishedOk := "DB_SCALE_CS_1".bo_CMD_FINISHED_OK,
                      i_boErr := "DB_SCALE_CS_1".bo_CMD_ERR,
                      io_iCmdInput := "DB_SCALE_CS_1".i_CMD_INPUT,
                      io_boEnable := "DB_SCALE_CS_1".bo_CMD_TRIGGER,
                      io_boAnyInProgress := "DB_SCALE_CS_1".bo_CMD_IN_PROGRESS,
                      io_stTask1 := "DB_SCALE_CS_1".s_CMD1,
                      io_stTask2 := "DB_SCALE_CS_1".s_CMD2,
                      io_stTask3 := "DB_SCALE_CS_1".s_CMD3);
END_REGION

REGION Network 4
   "FB_SICS_DR_T2"(ADDR := 280,   // "SICS_DR"
                   DB_SCALE := 62,
                   DB_VECTOR := 63,
                   CMD_IN := "DB_SCALE_CS_2".i_CMD_INPUT,
                   SEL_PROC_VAL := "DB_SCALE_CS_2".b_SELECT_PROC_VAL,
                   EXT_TARA := "DB_SCALE_CS_2".i_PRESET_TARE,
                   CMD_EN := "DB_SCALE_CS_2".bo_CMD_TRIGGER,
                   CMD_INPR => "DB_SCALE_CS_2".bo_CMD_IN_PROGRESS,
                   CMD_FOK => "DB_SCALE_CS_2".bo_CMD_FINISHED_OK,
                   CMD_ERR => "DB_SCALE_CS_2".bo_CMD_ERR,
                   CMD_ERR_C => "DB_SCALE_CS_2".b_CMD_ERR_CODE,
                   REF_COUNT => "DB_SCALE_CS_2".b_INFO_REFRESH_COUNT,
                   ACT_SEL_PROC_VAL => "DB_SCALE_CS_2".b_SELECTED_PROC_VAL,
                   PROC_VAL1 => "DB_SCALE_CS_2".i_PROCESS_VALUE,
                   SC_STATUS => "DB_SCALE_CS_2".w_SCALE_STATUS,
                   ERR_MSG_C => "DB_SCALE_CS_2".b_OPR_ERR_MSG,
                   FB_ERR => "DB_SCALE_CS_2".bo_FB_ERR,
                   FB_ERR_C => "DB_SCALE_CS_2".b_FB_ERR_CODE,
                   START_UP => "DB_SCALE_CS_2".bo_START_UP_IN_PROGRESS);
END_REGION

REGION Network 5
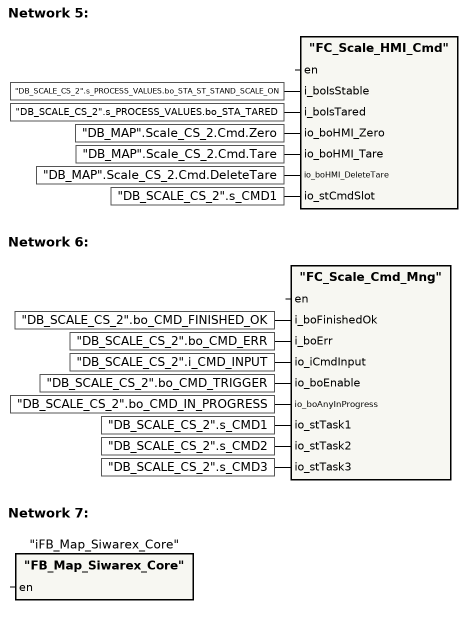
   "FC_Scale_HMI_Cmd"(i_boIsStable := "DB_SCALE_CS_2".s_PROCESS_VALUES.bo_STA_ST_STAND_SCALE_ON,
                      i_boIsTared := "DB_SCALE_CS_2".s_PROCESS_VALUES.bo_STA_TARED,
                      io_boHMI_Zero := "DB_MAP".Scale_CS_2.Cmd.Zero,
                      io_boHMI_Tare := "DB_MAP".Scale_CS_2.Cmd.Tare,
                      io_boHMI_DeleteTare := "DB_MAP".Scale_CS_2.Cmd.DeleteTare,
                      io_stCmdSlot := "DB_SCALE_CS_2".s_CMD1);
END_REGION

REGION Network 6
   "FC_Scale_Cmd_Mng"(i_boFinishedOk := "DB_SCALE_CS_2".bo_CMD_FINISHED_OK,
                      i_boErr := "DB_SCALE_CS_2".bo_CMD_ERR,
                      io_iCmdInput := "DB_SCALE_CS_2".i_CMD_INPUT,
                      io_boEnable := "DB_SCALE_CS_2".bo_CMD_TRIGGER,
                      io_boAnyInProgress := "DB_SCALE_CS_2".bo_CMD_IN_PROGRESS,
                      io_stTask1 := "DB_SCALE_CS_2".s_CMD1,
                      io_stTask2 := "DB_SCALE_CS_2".s_CMD2,
                      io_stTask3 := "DB_SCALE_CS_2".s_CMD3);
END_REGION

REGION Network 7
   "iFB_Map_Siwarex_Core"();   // "FB_Map_Siwarex_Core"
END_REGION
END_FUNCTION

FUNCTION "FC_Scale_HMI_Cmd" : Void
{ S7_Optimized_Access := 'FALSE' }
VERSION : 1.2
   VAR_INPUT 
      i_boIsStable : Bool;   // Статус модуля: Весы стабильны (Standstill)
      i_boIsTared : Bool;   // Статус модуля: Весы затарированы
   END_VAR

   VAR_IN_OUT 
      io_boHMI_Zero : Bool;   // Кнопка HMI: Обнулить
      io_boHMI_Tare : Bool;   // Кнопка HMI: Затарировать
      io_boHMI_DeleteTare : Bool;   // Кнопка HMI: Удалить тару
      io_stCmdSlot : "UDT_SIWA_Cmd";   // Слот задачи для передачи в менеджер (напр. sTask2)
   END_VAR


BEGIN
	    // =========================================================
	    // 1. Обнуление (Код 21)
	    // =========================================================
	    IF #io_boHMI_Zero THEN
	        IF #i_boIsStable AND NOT #io_stCmdSlot.bo_InProgress THEN
	            #io_stCmdSlot.i_Code := 21;
	            #io_stCmdSlot.bo_Trigger := TRUE;
	        END_IF;
	        #io_boHMI_Zero := FALSE;
	    END_IF;
	    
	    // =========================================================
	    // 2. Тарирование (Код 22)
	    // Защита от двойной тары (NOT i_boIsTared)
	    // =========================================================
	    IF #io_boHMI_Tare THEN
	        IF #i_boIsStable AND NOT #i_boIsTared AND NOT #io_stCmdSlot.bo_InProgress THEN
	            #io_stCmdSlot.i_Code := 22;
	            #io_stCmdSlot.bo_Trigger := TRUE;
	        END_IF;
	        #io_boHMI_Tare := FALSE;
	    END_IF;
	    
	    // =========================================================
	    // 3. Удаление тары (Код 24)
	    // =========================================================
	    IF #io_boHMI_DeleteTare THEN
	        IF #i_boIsTared AND NOT #io_stCmdSlot.bo_InProgress THEN
	            #io_stCmdSlot.i_Code := 24;
	            #io_stCmdSlot.bo_Trigger := TRUE;
	        END_IF;
	        #io_boHMI_DeleteTare := FALSE;
	    END_IF;
	    
END_FUNCTION

FUNCTION "FC_Scale_Cmd_Mng" : Void
{ S7_Optimized_Access := 'FALSE' }
VERSION : 1.6
   VAR_INPUT 
      i_boFinishedOk : Bool;   // Аппаратный статус: Команда завершена успешно
      i_boErr : Bool;   // Аппаратный статус: Ошибка выполнения
   END_VAR

   VAR_IN_OUT 
      io_iCmdInput : Int;   // Регистр команды модуля Siwarex
      io_boEnable : Bool;   // Триггер запуска аппаратной команды
      io_boAnyInProgress : Bool;   // Флаг: Модуль занят
      io_stTask1 : "UDT_SIWA_Cmd";   // Слот 1 (Высокий приоритет, напр. HMI)
      io_stTask2 : "UDT_SIWA_Cmd";   // Слот 2
      io_stTask3 : "UDT_SIWA_Cmd";   // Слот 3 (Низкий приоритет, напр. DR30)
   END_VAR


BEGIN
	    // 1. Очистка импульсных статусов
	    #io_stTask1.bo_FinishedOk := FALSE;
	    #io_stTask1.bo_FinishedError := FALSE;
	    
	    #io_stTask2.bo_FinishedOk := FALSE;
	    #io_stTask2.bo_FinishedError := FALSE;
	    
	    #io_stTask3.bo_FinishedOk := FALSE;
	    #io_stTask3.bo_FinishedError := FALSE;
	    
	    // 2. Проверка завершения текущей задачи
	    IF #io_boAnyInProgress THEN
	        IF #io_stTask1.bo_InProgress THEN
	            IF #i_boFinishedOk THEN
	                #io_stTask1.bo_FinishedOk := TRUE;
	            END_IF;
	            IF #i_boErr THEN
	                #io_stTask1.bo_FinishedError := TRUE;
	            END_IF;
	            
	            IF #i_boFinishedOk OR #i_boErr THEN
	                #io_stTask1.bo_InProgress := FALSE;
	                #io_boAnyInProgress := FALSE;
	                #io_boEnable := FALSE;
	            END_IF;
	            
	        ELSIF #io_stTask2.bo_InProgress THEN
	            IF #i_boFinishedOk THEN
	                #io_stTask2.bo_FinishedOk := TRUE;
	            END_IF;
	            IF #i_boErr THEN
	                #io_stTask2.bo_FinishedError := TRUE;
	            END_IF;
	            
	            IF #i_boFinishedOk OR #i_boErr THEN
	                #io_stTask2.bo_InProgress := FALSE;
	                #io_boAnyInProgress := FALSE;
	                #io_boEnable := FALSE;
	            END_IF;
	            
	        ELSIF #io_stTask3.bo_InProgress THEN
	            IF #i_boFinishedOk THEN
	                #io_stTask3.bo_FinishedOk := TRUE;
	            END_IF;
	            IF #i_boErr THEN
	                #io_stTask3.bo_FinishedError := TRUE;
	            END_IF;
	            
	            IF #i_boFinishedOk OR #i_boErr THEN
	                #io_stTask3.bo_InProgress := FALSE;
	                #io_boAnyInProgress := FALSE;
	                #io_boEnable := FALSE;
	            END_IF;
	        END_IF;
	    END_IF;
	    
	    // 3. Запуск новой задачи из очереди (по приоритету 1 -> 2 -> 3)
	    IF NOT #io_boAnyInProgress AND NOT #io_boEnable THEN
	        IF #io_stTask1.bo_Trigger THEN
	            #io_iCmdInput := #io_stTask1.i_Code;
	            #io_stTask1.bo_InProgress := TRUE;
	            #io_boAnyInProgress := TRUE;
	            #io_boEnable := TRUE;
	            #io_stTask1.bo_Trigger := FALSE;
	            
	        ELSIF #io_stTask2.bo_Trigger THEN
	            #io_iCmdInput := #io_stTask2.i_Code;
	            #io_stTask2.bo_InProgress := TRUE;
	            #io_boAnyInProgress := TRUE;
	            #io_boEnable := TRUE;
	            #io_stTask2.bo_Trigger := FALSE;
	            
	        ELSIF #io_stTask3.bo_Trigger THEN
	            #io_iCmdInput := #io_stTask3.i_Code;
	            #io_stTask3.bo_InProgress := TRUE;
	            #io_boAnyInProgress := TRUE;
	            #io_boEnable := TRUE;
	            #io_stTask3.bo_Trigger := FALSE;
	        END_IF;
	    END_IF;
END_FUNCTION

FUNCTION_BLOCK "FB_Map_Siwarex_Core"
TITLE = Маппинг данных Siwarex CS
{ S7_Optimized_Access := 'FALSE' }
AUTHOR : S7C_Lib
FAMILY : Analog
VERSION : 1.4
// ==============================================================================
// Описание: Адаптированный маппинг из UDT_SIWA_CS. Обработка раздельных кодов 
//           ошибок (модуля и драйвера). Встроенный таймер Watchdog в STAT.
// ==============================================================================
   VAR_INPUT 
      i_Scale_DB : "UDT_SIWA_CS";   // Системный интерфейс Siwarex CS
      i_CycleTime_ms : Int;   // Время цикла ПЛК для таймера Watchdog
   END_VAR

   VAR_IN_OUT 
      io_Core : "UDT_Siwarex_Core";   // Плоская структура
   END_VAR

   VAR 
      stat_Diag : Struct   // Внутренняя память для Watchdog
         Old_Count : Byte;
         Old_Weight : Real;
         Last_Change_ms : DInt;
      END_STRUCT;
   END_VAR

   VAR_TEMP 
      temp_Value_Changed : Bool;
      temp_Counter_Changed : Bool;
   END_VAR


BEGIN
	    // 1. Веса
	    #io_Core.Weight_Gross_kg := INT_TO_REAL(#i_Scale_DB.s_PROCESS_VALUES.i_GROSS_WEIGHT_PROC);
	    #io_Core.Weight_Net_kg := INT_TO_REAL(#i_Scale_DB.s_PROCESS_VALUES.i_NET_WEIGHT_PROC);
	    #io_Core.Weight_Tare_kg := INT_TO_REAL(#i_Scale_DB.s_PROCESS_VALUES.i_TARE_WEIGHT_PROC);
	    
	    // 2. Диагностика (Коды ошибок) - извлекаем типы Byte в Int
	    // Операционная ошибка
	    #io_Core.Error_Op_Msg := BYTE_TO_INT(#i_Scale_DB.s_PROCESS_VALUES.b_OPR_ERR_MSG);
	    // Ошибка драйвера
	    #io_Core.Error_FB_Code := BYTE_TO_INT(#i_Scale_DB.b_FB_ERR_CODE);
	    
	    // 3. Диагностика (Биты)
	    #io_Core.Status.Standstill := #i_Scale_DB.s_PROCESS_VALUES.bo_STA_ST_STAND_SCALE_ON;
	    #io_Core.Status.Limit_1 := #i_Scale_DB.s_PROCESS_VALUES.bo_STA_LIMIT1_ON;
	    #io_Core.Status.Limit_2 := #i_Scale_DB.s_PROCESS_VALUES.bo_STA_LIMIT2_ON;
	    #io_Core.Status.Fault_HW := #i_Scale_DB.s_PROCESS_VALUES.bo_STA_ERROR_ON;
	    #io_Core.Status.Limit_Max := #i_Scale_DB.s_PROCESS_VALUES.bo_STA_MAX_9E;
	    #io_Core.Status.Fault_FB := #i_Scale_DB.bo_FB_ERR; // Флаг ошибки FB
	    
	    // 4. Логика Watchdog (Контроль зависания)
	    #temp_Value_Changed := (#io_Core.Weight_Net_kg <> #stat_Diag.Old_Weight);
	    #temp_Counter_Changed := (#i_Scale_DB.b_INFO_REFRESH_COUNT <> #stat_Diag.Old_Count);
	    
	    IF #temp_Value_Changed OR #temp_Counter_Changed THEN
	        #stat_Diag.Last_Change_ms := 0;
	        #stat_Diag.Old_Weight := #io_Core.Weight_Net_kg;
	        #stat_Diag.Old_Count := #i_Scale_DB.b_INFO_REFRESH_COUNT;
	        #io_Core.Status.Comm_Fault := FALSE;
	    ELSE
	        #stat_Diag.Last_Change_ms := #stat_Diag.Last_Change_ms + INT_TO_DINT(#i_CycleTime_ms);
	    END_IF;
	    
	    IF #stat_Diag.Last_Change_ms > 5000 THEN
	        #io_Core.Status.Comm_Fault := TRUE;
	    END_IF;
	    
END_FUNCTION_BLOCK

FUNCTION_BLOCK "FB_Sim_SawTooth"
{ S7_Optimized_Access := 'FALSE' }
VERSION : 0.1
   VAR_INPUT 
      Enable : Bool;
      Speed : Real;
   END_VAR

   VAR_OUTPUT 
      Out_Raw : Int;
   END_VAR

   VAR 
      Current_Val : Real;
   END_VAR


BEGIN
	
	IF NOT #Enable THEN
	    #Current_Val := 0.0;
	    #Out_Raw := 0;
	    RETURN;
	END_IF;
	#Current_Val := #Current_Val + (#Speed * "getCycleTime"() / 1000.0);
	IF #Current_Val > 27648.0 THEN
	    #Current_Val := 0.0;
	END_IF;
	#Out_Raw := REAL_TO_INT(#Current_Val);
	
END_FUNCTION_BLOCK

FUNCTION "FC_ScaleValue" : Real
{ S7_Optimized_Access := 'FALSE' }
VERSION : 0.1
// 4. LIBRARY FUNCTIONS (FC_ScaleValue, FC_Filter_PT1 from previous turns)
   VAR_INPUT 
      i_rInp : Real;
      i_rInpLow : Real;
      i_rInpHigh : Real;
      i_rOutLow : Real;
      i_rOutHigh : Real;
      i_boUseLimit : Bool;
      i_boUseSqrt : Bool;
      i_rCutoff : Real;
   END_VAR

   VAR_TEMP 
      temp_rNorm : Real;
      temp_rResult : Real;
   END_VAR


BEGIN
	
	IF ABS(#i_rInpHigh - #i_rInpLow) < 0.000001 THEN
	    #FC_ScaleValue := #i_rOutLow;
	    RETURN;
	END_IF;
	#temp_rNorm := (#i_rInp - #i_rInpLow) / (#i_rInpHigh - #i_rInpLow);
	IF #i_boUseSqrt THEN
	    IF #temp_rNorm < 0.0 THEN
	        #temp_rNorm := 0.0;
	    END_IF;
	    #temp_rNorm := SQRT(#temp_rNorm);
	END_IF;
	#temp_rResult := (#temp_rNorm * (#i_rOutHigh - #i_rOutLow)) + #i_rOutLow;
	IF ABS(#temp_rResult - #i_rOutLow) <= ABS(#i_rCutoff) THEN
	    #temp_rResult := #i_rOutLow;
	END_IF;
	IF #i_boUseLimit THEN
	    IF #i_rOutHigh > #i_rOutLow THEN
	        IF #temp_rResult > #i_rOutHigh THEN
	            #temp_rResult := #i_rOutHigh;
	        END_IF;
	        IF #temp_rResult < #i_rOutLow THEN
	            #temp_rResult := #i_rOutLow;
	        END_IF;
	    ELSE
	        IF #temp_rResult < #i_rOutHigh THEN
	            #temp_rResult := #i_rOutHigh;
	        END_IF;
	        IF #temp_rResult > #i_rOutLow THEN
	            #temp_rResult := #i_rOutLow;
	        END_IF;
	    END_IF;
	END_IF;
	#FC_ScaleValue := #temp_rResult;
	
END_FUNCTION

FUNCTION_BLOCK "FB_DI"
TITLE = Func Block from DI
{ S7_Optimized_Access := 'FALSE' }
VERSION : 1.2
// ==============================================================================
// Файл: S7C_FC_Filter_PT1.scl
// Целевые ПЛК: S7-1200 / S7-1500 (Линейка Current)
// Особенности: 
// - Оптимизированный доступ (Optimized block access = TRUE)
// - Использование современных системных функций (время цикла, первый скан)
// - Кодировка при сохранении: UTF-8 with BOM
// ==============================================================================
   VAR_INPUT 
      i_boRaw : Bool;   // Сырой физический вход
   END_VAR

   VAR_IN_OUT 
      io_stConfig : "UDT_DI_Conf";
      io_stOut : "UDT_DI_Out";
   END_VAR

   VAR 
      stat_TonFlt {InstructionName := 'TON'; LibVersion := '1.0'; S7_SetPoint := 'False'} : TON;   // Задержка включения
      stat_TofFlt {InstructionName := 'TOF'; LibVersion := '1.0'; S7_SetPoint := 'False'} : TOF;   // Задержка выключения
      stat_Mode : Int;   // Текущий рабочий режим
      stat_OldMode : Int;   // Предыдущий режим для отслеживания изменений
   END_VAR

   VAR_TEMP 
      temp_FilterTime : Time;
   END_VAR


BEGIN
	    // =========================================================
	    // 1. ПРОВЕРКА РЕЖИМА И ПРЕОБРАЗОВАНИЕ ВРЕМЕНИ
	    // =========================================================
	    IF #io_stConfig.Mode > 2 OR #io_stConfig.Mode < 0 THEN
	        #stat_Mode := 0;
	    ELSE
	        #stat_Mode := #io_stConfig.Mode;
	    END_IF;
	    
	    // Преобразуем мс (Int) в формат Time
	    #temp_FilterTime := DINT_TO_TIME(INT_TO_DINT(#io_stConfig.FilterTime));
	    
	    // =========================================================
	    // 2. СБРОС ТАЙМЕРОВ ПРИ СМЕНЕ РЕЖИМА
	    // =========================================================
	    IF #stat_Mode <> #stat_OldMode THEN
	        #stat_TonFlt(IN := FALSE,
	                     PT := #temp_FilterTime);
	        #stat_TofFlt(IN := FALSE,
	                     PT := #temp_FilterTime);
	        
	        #io_stOut.Value := #i_boRaw;
	        #stat_OldMode := #stat_Mode;
	    END_IF;
	    
	    // =========================================================
	    // 3. ЛОГИКА ФИЛЬТРАЦИИ И ИНВЕРСИИ
	    // =========================================================
	    IF #stat_Mode = 0 THEN
	        // Режим 0: Прямая передача сигнала (без фильтра)
	        #io_stOut.Value := #i_boRaw;
	        
	        // Сбрасываем таймеры, чтобы они не висели в фоне
	        #stat_TonFlt(IN := FALSE,
	                     PT := #temp_FilterTime);
	        #stat_TofFlt(IN := FALSE,
	                     PT := #temp_FilterTime);
	        
	    ELSE
	        // Режимы с фильтром: применяем TON и TOF
	        #stat_TonFlt(IN := #i_boRaw,
	                     PT := #temp_FilterTime);
	        #stat_TofFlt(IN := #i_boRaw,
	                     PT := #temp_FilterTime);
	        
	        // Включение (TON отработал) -> сигнал стабильно TRUE
	        IF #stat_TonFlt.Q THEN
	            #io_stOut.Value := (#stat_Mode = 1); // 1 = Прямой, 2 = Инверсный
	        END_IF;
	        
	        // Выключение (TOF отработал) -> сигнал стабильно FALSE
	        IF NOT #stat_TofFlt.Q THEN
	            #io_stOut.Value := (#stat_Mode <> 1); // Сбрасываем соответственно режиму
	        END_IF;
	    END_IF;
	    
END_FUNCTION_BLOCK

FUNCTION_BLOCK "FB_DI_Alarm"
{ S7_Optimized_Access := 'FALSE' }
VERSION : 1.0
// =============================================================================
// БЛОК ДИСКРЕТНОГО АЛАРМА
// =============================================================================
   VAR_INPUT 
      i_boSignal : Bool;   // Обработанный сигнал (от FB_DI)
      i_boReset : Bool;   // Команда сброса (Квитирование)
      i_boInhibit : Bool;   // Блокировка (например, при потере питания шкафа)
   END_VAR

   VAR_IN_OUT 
      io_stConfig : "UDT_DI_Alarm_Conf";
      io_stOut : "UDT_DI_Alarm";
   END_VAR

   VAR 
      stat_TonAlarm {InstructionName := 'TON'; LibVersion := '1.0'; S7_SetPoint := 'False'} : TON;   // Таймер задержки срабатывания
      stat_InputInv : Bool;   // Внутренний статус после учета инверсии
   END_VAR


BEGIN
	    // =========================================================
	    // 1. ТРАНСЛЯЦИЯ СТАТУСОВ ДЛЯ HMI (En_Out)
	    // =========================================================
	    #io_stOut.En_Alarm := #io_stConfig.En_Alarm AND NOT #i_boInhibit;
	    #io_stOut.Latch_Enable := #io_stConfig.Latch_Enable;
	    #io_stOut.Input_Raw := #i_boSignal;
	    
	    // =========================================================
	    // 2. ИНВЕРСИЯ СИГНАЛА (XOR)
	    // =========================================================
	    // Если Invert=0: Авария наступает при Signal=TRUE (замыкание)
	    // Если Invert=1: Авария наступает при Signal=FALSE (размыкание)
	    #stat_InputInv := #i_boSignal XOR #io_stConfig.Invert;
	    #io_stOut.Input_Inv := #stat_InputInv;
	    
	    // =========================================================
	    // 3. ТАЙМЕР ЗАДЕРЖКИ (В СЕКУНДАХ)
	    // =========================================================
	    // Вычисляем время и передаем в таймер. Если Inhibit активен или аларм выключен - таймер сбрасывается.
	    #stat_TonAlarm(IN := #stat_InputInv AND #io_stOut.En_Alarm,
	                   PT := DINT_TO_TIME(INT_TO_DINT(#io_stConfig.Delay)) * 1000);
	    
	    // =========================================================
	    // 4. ЛОГИКА ФИКСАЦИИ (LATCH) И СБРОСА
	    // =========================================================
	    // Сброс происходит, если:
	    // 1. Сработала внешняя блокировка (Inhibit)
	    // 2. Авария выключена в конфигурации
	    // 3. Сигнал в норме И (нет фиксации ИЛИ нажата кнопка сброса)
	    
	    IF #i_boInhibit OR NOT #io_stConfig.En_Alarm OR
	        (NOT #stat_InputInv AND (NOT #io_stConfig.Latch_Enable OR #i_boReset)) THEN
	        #io_stOut.Alarm := FALSE;
	    ELSIF #stat_TonAlarm.Q THEN
	        #io_stOut.Alarm := TRUE;
	    END_IF;
	    
END_FUNCTION_BLOCK

FUNCTION "FC_Tank_Calc" : Void
TITLE = Syrup Tank Physics
{ S7_Optimized_Access := 'FALSE' }
AUTHOR : Gemini
FAMILY : Archive
VERSION : 1.1
   VAR_INPUT 
      i_rValue : Real;   // Входящее значение (мм или кг)
      i_boIsSiwa : Bool;   // TRUE = Весы (кг), FALSE = Уровень (мм)
   END_VAR

   VAR_IN_OUT 
      io_Geom : "UDT_Tank_Geom";
      iq_Calc : "UDT_Tank_Calc";
   END_VAR

   VAR_TEMP 
      temp_rDensity : Real;
      temp_rMaxVol : Real;
      temp_rHeight : Real;
   END_VAR


BEGIN
	    // Предотвращение деления на ноль (Safety Check)
	    IF #io_Geom.Density < 0.1 THEN
	        #temp_rDensity := 1000.0;
	    ELSE
	        #temp_rDensity := #io_Geom.Density;
	    END_IF;
	    IF #io_Geom.Max_Volume < 0.1 THEN
	        #temp_rMaxVol := 1.0;
	    ELSE
	        #temp_rMaxVol := #io_Geom.Max_Volume;
	    END_IF;
	    IF #io_Geom.Height_Full < 0.1 THEN
	        #temp_rHeight := 1.0;
	    ELSE
	        #temp_rHeight := #io_Geom.Height_Full;
	    END_IF;
	    
	    IF #i_boIsSiwa THEN
	        // --- РЕЖИМ ВЕСОВ (Siwarex) ---
	        #iq_Calc.Weight_t := #i_rValue / 1000.0; // кг -> т
	        #iq_Calc.Volume_m3 := #i_rValue / #temp_rDensity; // V = m / rho
	        
	        // Обратный расчет уровня для визуализации
	        #iq_Calc.Level_Pct := (#iq_Calc.Volume_m3 / #temp_rMaxVol) * 100.0;
	        #iq_Calc.Level_m := (#iq_Calc.Level_Pct * #temp_rHeight) / 100.0;
	    ELSE
	        // --- РЕЖИМ УРОВНЯ (4-20 мА) ---
	        #iq_Calc.Level_m := #i_rValue + #io_Geom.Sensor_Offset;
	        #iq_Calc.Level_Pct := (#iq_Calc.Level_m / #temp_rHeight) * 100.0;
	        
	        // Расчет объема и веса
	        #iq_Calc.Volume_m3 := (#temp_rMaxVol * #iq_Calc.Level_Pct) / 100.0;
	        #iq_Calc.Weight_t := (#iq_Calc.Volume_m3 * #temp_rDensity) / 1000.0;
	    END_IF;
	    
	    // Свободное место
	    #iq_Calc.Ullage_m3 := #temp_rMaxVol - #iq_Calc.Volume_m3;
	    IF #iq_Calc.Ullage_m3 < 0.0 THEN
	        #iq_Calc.Ullage_m3 := 0.0;
	    END_IF;
	    
END_FUNCTION

FUNCTION_BLOCK "FB_AI_Alarm"
{ S7_Optimized_Access := 'FALSE' }
VERSION : 2.0
   VAR_INPUT 
      i_rValue : Real;
      i_boReset : Bool;
      i_boInhibit : Bool;
   END_VAR

   VAR_IN_OUT 
      io_stConfig : "UDT_AI_Alarm_Conf";
      io_stOut : "UDT_AI_Alarm";
   END_VAR

   VAR 
      stat_TonHiHi {InstructionName := 'TON'; LibVersion := '1.0'; S7_SetPoint := 'False'} : TON;
      stat_TonHi {InstructionName := 'TON'; LibVersion := '1.0'; S7_SetPoint := 'False'} : TON;
      stat_TonLo {InstructionName := 'TON'; LibVersion := '1.0'; S7_SetPoint := 'False'} : TON;
      stat_TonLoLo {InstructionName := 'TON'; LibVersion := '1.0'; S7_SetPoint := 'False'} : TON;
      stat_RawHiHi : Bool;
      stat_RawHi : Bool;
      stat_RawLo : Bool;
      stat_RawLoLo : Bool;
   END_VAR


BEGIN
	    // =========================================================
	    // 0. ЗАЩИТА ОТ ДУРАКА (Ограничение уставок времени >= 0)
	    // =========================================================
	    IF #io_stConfig.Delay_HiHi < 0 THEN
	        #io_stConfig.Delay_HiHi := 0;
	    END_IF;
	    IF #io_stConfig.Delay_Hi < 0 THEN
	        #io_stConfig.Delay_Hi := 0;
	    END_IF;
	    IF #io_stConfig.Delay_Lo < 0 THEN
	        #io_stConfig.Delay_Lo := 0;
	    END_IF;
	    IF #io_stConfig.Delay_LoLo < 0 THEN
	        #io_stConfig.Delay_LoLo := 0;
	    END_IF;
	    
	    // =========================================================
	    // 1. ТРАНСЛЯЦИЯ СТАТУСОВ ДЛЯ HMI (En_Out)
	    // =========================================================
	    #io_stOut.En_HiHi := #io_stConfig.En_Alarm.HiHi AND NOT #i_boInhibit;
	    #io_stOut.En_Hi := #io_stConfig.En_Alarm.Hi AND NOT #i_boInhibit;
	    #io_stOut.En_Lo := #io_stConfig.En_Alarm.Lo AND NOT #i_boInhibit;
	    #io_stOut.En_LoLo := #io_stConfig.En_Alarm.LoLo AND NOT #i_boInhibit;
	    #io_stOut.En_Latch_Enable := #io_stConfig.En_Alarm.Latch_Enable;
	    
	    // =========================================================
	    // 2. ОБРАБОТКА СЫРЫХ АВАРИЙ С ГИСТЕРЕЗИСОМ (Deadband)
	    // =========================================================
	    // Верхние пороги (Срабатывание >, Сброс <)
	    IF #i_rValue > #io_stConfig.HiHi THEN
	        #stat_RawHiHi := TRUE;
	    ELSIF #i_rValue < (#io_stConfig.HiHi - #io_stConfig.Hysteresis) THEN
	        #stat_RawHiHi := FALSE;
	    END_IF;
	    
	    IF #i_rValue > #io_stConfig.Hi THEN
	        #stat_RawHi := TRUE;
	    ELSIF #i_rValue < (#io_stConfig.Hi - #io_stConfig.Hysteresis) THEN
	        #stat_RawHi := FALSE;
	    END_IF;
	    
	    // Нижние пороги (Срабатывание <, Сброс >)
	    IF #i_rValue < #io_stConfig.Lo THEN
	        #stat_RawLo := TRUE;
	    ELSIF #i_rValue > (#io_stConfig.Lo + #io_stConfig.Hysteresis) THEN
	        #stat_RawLo := FALSE;
	    END_IF;
	    
	    IF #i_rValue < #io_stConfig.LoLo THEN
	        #stat_RawLoLo := TRUE;
	    ELSIF #i_rValue > (#io_stConfig.LoLo + #io_stConfig.Hysteresis) THEN
	        #stat_RawLoLo := FALSE;
	    END_IF;
	    
	    // =========================================================
	    // 3. ТАЙМЕРЫ ЗАДЕРЖКИ (ON-Delay)
	    // =========================================================
	    // Таймер не считает, если сработала блокировка датчика (Inhibit) 
	    // или аларм выключен в настройках.
	    #stat_TonHiHi(IN := #stat_RawHiHi AND #io_stConfig.En_Alarm.HiHi AND NOT #i_boInhibit,
	                  PT := DINT_TO_TIME(#io_stConfig.Delay_HiHi) * 1000 + t#1ms);//gr-ny 300
	    
	    #stat_TonHi(IN := #stat_RawHi AND #io_stConfig.En_Alarm.Hi AND NOT #i_boInhibit,
	                PT := DINT_TO_TIME(#io_stConfig.Delay_Hi) * 1000 + t#1ms);//gr-ny 300
	    
	    #stat_TonLo(IN := #stat_RawLo AND #io_stConfig.En_Alarm.Lo AND NOT #i_boInhibit,
	                PT := DINT_TO_TIME(#io_stConfig.Delay_Lo) * 1000 + t#1ms);//gr-ny 300
	    
	    #stat_TonLoLo(IN := #stat_RawLoLo AND #io_stConfig.En_Alarm.LoLo AND NOT #i_boInhibit,
	                  PT := DINT_TO_TIME(#io_stConfig.Delay_LoLo) * 1000 + t#1ms);//gr-ny 300
	    
	    // =========================================================
	    // 4. ФИКСАЦИЯ (LATCH) И СБРОС АВАРИЙ
	    // =========================================================
	    // Логика сброса (имеет приоритет):
	    // 1. Сработал Inhibit (глушим всё безусловно)
	    // 2. Аларм сняли в настройках
	    // 3. Уровень в норме И (нет фиксации ИЛИ нажата кнопка Reset)
	    
	    // --- HiHi ---
	    IF #i_boInhibit OR NOT #io_stConfig.En_Alarm.HiHi OR
	        (NOT #stat_RawHiHi AND (NOT #io_stConfig.En_Alarm.Latch_Enable OR #i_boReset)) THEN
	        #io_stOut.HiHi := FALSE;
	    ELSIF #stat_TonHiHi.Q THEN
	        #io_stOut.HiHi := TRUE;
	    END_IF;
	    
	    // --- Hi ---
	    IF #i_boInhibit OR NOT #io_stConfig.En_Alarm.Hi OR
	        (NOT #stat_RawHi AND (NOT #io_stConfig.En_Alarm.Latch_Enable OR #i_boReset)) THEN
	        #io_stOut.Hi := FALSE;
	    ELSIF #stat_TonHi.Q THEN
	        #io_stOut.Hi := TRUE;
	    END_IF;
	    
	    // --- Lo ---
	    IF #i_boInhibit OR NOT #io_stConfig.En_Alarm.Lo OR
	        (NOT #stat_RawLo AND (NOT #io_stConfig.En_Alarm.Latch_Enable OR #i_boReset)) THEN
	        #io_stOut.Lo := FALSE;
	    ELSIF #stat_TonLo.Q THEN
	        #io_stOut.Lo := TRUE;
	    END_IF;
	    
	    // --- LoLo ---
	    IF #i_boInhibit OR NOT #io_stConfig.En_Alarm.LoLo OR
	        (NOT #stat_RawLoLo AND (NOT #io_stConfig.En_Alarm.Latch_Enable OR #i_boReset)) THEN
	        #io_stOut.LoLo := FALSE;
	    ELSIF #stat_TonLoLo.Q THEN
	        #io_stOut.LoLo := TRUE;
	    END_IF;
	    
END_FUNCTION_BLOCK

FUNCTION_BLOCK "FB_Time_Trigger"
TITLE = 'Генератор часовых слепков (Пуленепробиваемый)'
{ S7_Optimized_Access := 'FALSE' }
AUTHOR : S7A_Lib
FAMILY : Archive
VERSION : 1.1
   VAR_INPUT 
      i_Shift_1_Start { ExternalAccessible := 'False'; ExternalVisible := 'False'; ExternalWritable := 'False'} : Int := 8;   // Час начала дневной смены (напр. 08:00)
      i_Shift_2_Start { ExternalAccessible := 'False'; ExternalVisible := 'False'; ExternalWritable := 'False'} : Int := 20;   // Час начала ночной смены (напр. 20:00)
   END_VAR

   VAR_OUTPUT 
      q_Trigger_Hour { ExternalAccessible := 'False'; ExternalVisible := 'False'; ExternalWritable := 'False'} : Bool;   // Импульс: Сменился час (или день)
      q_Trigger_Shift { ExternalAccessible := 'False'; ExternalVisible := 'False'; ExternalWritable := 'False'} : Bool;   // Импульс: Началась новая смена
   END_VAR

   VAR 
      stat_Prev_Hour { ExternalAccessible := 'False'; ExternalVisible := 'False'; ExternalWritable := 'False'} : Int;
      stat_Prev_Day { ExternalAccessible := 'False'; ExternalVisible := 'False'; ExternalWritable := 'False'} : Int;   // ДОБАВЛЕНО: Память предыдущего дня
      stat_Init_Done { ExternalAccessible := 'False'; ExternalVisible := 'False'; ExternalWritable := 'False'} : Bool;
      temp_DT { ExternalAccessible := 'False'; ExternalVisible := 'False'; ExternalWritable := 'False'} : Date_And_Time;
      temp_DT_Bytes { ExternalAccessible := 'False'; ExternalVisible := 'False'; ExternalWritable := 'False'} AT temp_DT : Array[0..7] of Byte;
      temp_Second_Int { ExternalAccessible := 'False'; ExternalVisible := 'False'; ExternalWritable := 'False'} : Int;
      temp_Minute_Int { ExternalAccessible := 'False'; ExternalVisible := 'False'; ExternalWritable := 'False'} : Int;
      temp_Hour_Int { ExternalAccessible := 'False'; ExternalVisible := 'False'; ExternalWritable := 'False'} : Int;
      temp_Day_Int { ExternalAccessible := 'False'; ExternalVisible := 'False'; ExternalWritable := 'False'} : Int;   // ДОБАВЛЕНО: Текущий день
      temp_Month_Int { ExternalAccessible := 'False'; ExternalVisible := 'False'; ExternalWritable := 'False'} : Int;
      temp_Yar_Int { ExternalAccessible := 'False'; ExternalVisible := 'False'; ExternalWritable := 'False'} : Int;
      temp_RetVal { ExternalAccessible := 'False'; ExternalVisible := 'False'; ExternalWritable := 'False'} : Int;
   END_VAR


BEGIN
	    #q_Trigger_Hour := FALSE;
	    #q_Trigger_Shift := FALSE;
	    
	    #temp_RetVal := RD_SYS_T(OUT => #temp_DT);
	    
	    #temp_Second_Int := BCD16_TO_INT(BYTE_TO_WORD(#temp_DT_Bytes[5]));
	    #temp_Minute_Int := BCD16_TO_INT(BYTE_TO_WORD(#temp_DT_Bytes[4]));
	    #temp_Hour_Int := BCD16_TO_INT(BYTE_TO_WORD(#temp_DT_Bytes[3]));
	    
	    #temp_Day_Int := BCD16_TO_INT(BYTE_TO_WORD(#temp_DT_Bytes[2]));
	    #temp_Month_Int := BCD16_TO_INT(BYTE_TO_WORD(#temp_DT_Bytes[1]));
	    #temp_Yar_Int := BCD16_TO_INT(BYTE_TO_WORD(#temp_DT_Bytes[0]));
	    
	    "DB_DateTime".DT_Byte := #temp_DT_Bytes;
	    "DB_DateTime".DateTime_PLC := #temp_DT;
	    "DB_DateTime".Date_PLC := DT_TO_DATE(#temp_DT);
	    "DB_DateTime".TimeOfDay_PLC := DT_TO_TOD(#temp_DT);
	    
	    // Инициализация при первой заливке блока
	    IF NOT #stat_Init_Done THEN
	        #stat_Prev_Hour := #temp_Hour_Int;
	        #stat_Prev_Day := #temp_Day_Int;
	        #stat_Init_Done := TRUE;
	        #q_Trigger_Hour := TRUE;
	        RETURN;
	    END_IF;
	    
	    // Контроль смены часа ИЛИ смены дня (закрывает баг "ровно 24 часа")
	    IF (#temp_Hour_Int <> #stat_Prev_Hour) OR (#temp_Day_Int <> #stat_Prev_Day) THEN
	        
	        #q_Trigger_Hour := TRUE;
	        
	        // Проверяем на начало смены
	        IF (#temp_Hour_Int = #i_Shift_1_Start) OR (#temp_Hour_Int = #i_Shift_2_Start) THEN
	            #q_Trigger_Shift := TRUE;
	        END_IF;
	        
	        // Обновляем память
	        #stat_Prev_Hour := #temp_Hour_Int;
	        #stat_Prev_Day := #temp_Day_Int;
	        
	    END_IF;
	    
END_FUNCTION_BLOCK

ORGANIZATION_BLOCK "COMPLETE RESTART"
TITLE = "Complete Restart"
{ S7_Optimized_Access := 'FALSE' }
VERSION : 0.1
   VAR_TEMP 
      OB100_EV_CLASS : Byte;   // 16#13, Event class 1, Entering event state, Event logged in diagnostic buffer
      OB100_STRTUP : Byte;   // 16#81/82/83/84 Method of startup
      OB100_PRIORITY : Byte;   // Priority of OB Execution
      OB100_OB_NUMBR : Byte;   // 100 (Organization block 100, OB100)
      OB100_RESERVED_1 : Byte;   // Reserved for system
      OB100_RESERVED_2 : Byte;   // Reserved for system
      OB100_STOP : Word;   // Event that caused CPU to stop (16#4xxx)
      OB100_STRT_INFO : DWord;   // Information on how system started
      OB100_DATE_TIME : Date_And_Time;   // Date and time OB100 started
   END_VAR


BEGIN
	
	"FC_ResetScaleCmd"();
END_ORGANIZATION_BLOCK

FUNCTION "FC_ResetScaleCmd" : Void
{ S7_Optimized_Access := 'FALSE' }
VERSION : 0.1
   VAR_TEMP 
      tmp_Cmd : "UDT_SIWA_Cmd";
      tmp_Cmd_Raw AT tmp_Cmd : Array[0..3] of Byte;
   END_VAR


BEGIN
	// Зачищаем все 4 байта включая паддинг
	#tmp_Cmd_Raw[0] := 16#00;
	#tmp_Cmd_Raw[1] := 16#00;
	#tmp_Cmd_Raw[2] := 16#00;
	#tmp_Cmd_Raw[3] := 16#00;
	
	// Применяем ко всем слотам обоих модулей
	"DB_SCALE_CS_1".s_CMD1 := #tmp_Cmd;
	"DB_SCALE_CS_1".s_CMD2 := #tmp_Cmd;
	"DB_SCALE_CS_1".s_CMD3 := #tmp_Cmd;
	
	"DB_SCALE_CS_2".s_CMD1 := #tmp_Cmd;
	"DB_SCALE_CS_2".s_CMD2 := #tmp_Cmd;
	"DB_SCALE_CS_2".s_CMD3 := #tmp_Cmd;
END_FUNCTION

ORGANIZATION_BLOCK "CYC_INT5"
TITLE = "Cyclic Interrupt"
{ S7_Optimized_Access := 'FALSE' }
VERSION : 0.1
   VAR_TEMP 
      OB35_EV_CLASS : Byte;   // Bits 0-3 = 1 (Coming event), Bits 4-7 = 1 (Event class 1)
      OB35_STRT_INF : Byte;   // 16#36 (OB 35 has started)
      OB35_PRIORITY : Byte;   // Priority of OB Execution
      OB35_OB_NUMBR : Byte;   // 35 (Organization block 35, OB35)
      OB35_RESERVED_1 : Byte;   // Reserved for system
      OB35_RESERVED_2 : Byte;   // Reserved for system
      OB35_PHASE_OFFSET : Word;   // Phase offset (msec)
      OB35_RESERVED_3 : Int;   // Reserved for system
      OB35_EXC_FREQ : Int;   // Frequency of execution (msec)
      OB35_DATE_TIME : Date_And_Time;   // Date and time OB35 started
   END_VAR


BEGIN
	// Опрос Танка 1 (Слот 3 - фоновое чтение веса)
	"FC_Weighing_Poll"(
	                   i_boAnyInProgress := "DB_SCALE_CS_1".bo_CMD_IN_PROGRESS,
	                   i_boCmdEnable     := "DB_SCALE_CS_1".bo_CMD_TRIGGER,
	                   io_stTask          := "DB_SCALE_CS_1".s_CMD3
	);
	
	// Опрос Танка 2 (Слот 3 - фоновое чтение веса)
	"FC_Weighing_Poll"(
	                   i_boAnyInProgress := "DB_SCALE_CS_2".bo_CMD_IN_PROGRESS,
	                   i_boCmdEnable     := "DB_SCALE_CS_2".bo_CMD_TRIGGER,
	                   io_stTask          := "DB_SCALE_CS_2".s_CMD3
	);
END_ORGANIZATION_BLOCK

FUNCTION "FC_Weighing_Poll" : Void
{ S7_Optimized_Access := 'FALSE' }
VERSION : 1.2
   VAR_INPUT 
      i_boAnyInProgress : Bool;   // Общий статус занятости модуля
      i_boCmdEnable : Bool;   // Общий триггер команд модуля
   END_VAR

   VAR_IN_OUT 
      io_stTask : "UDT_SIWA_Cmd";   // Слот задачи циклического опроса (напр. sTask3)
   END_VAR


BEGIN
	    // ===================================================
	    // Генерация команды чтения Data Record (DR30 - Код 230)
	    // Функция предназначена для циклического вызова (OB35)
	    // ===================================================
	    IF NOT #i_boAnyInProgress AND NOT #i_boCmdEnable AND NOT #io_stTask.bo_InProgress THEN
	        #io_stTask.i_Code := 230;
	        #io_stTask.bo_Trigger := TRUE;
	    END_IF;
	    
END_FUNCTION

FUNCTION "Formula_weight_tank" : Void
{ S7_Optimized_Access := 'FALSE' }
VERSION : 0.1
   VAR_INPUT 
      S : Real;
      P : Real;
      Den : Real;
   END_VAR

   VAR_IN_OUT 
      P_z : Real;
      P_w : Real;
      Zero_But : Bool;
      Weight_But : Bool;
      Weight : Real;
      Weight_zero : Real;
      Weight_DB : Real;
      Korect : Bool;
   END_VAR


BEGIN
	#Weight := (#S * ((#P / (9.81 * #Den)) * 100)) * #Den;
	
	IF #Zero_But = TRUE
	THEN
	    #Weight_zero := #Weight;
	    #P_z := #P;
	    #Zero_But := FALSE;
	END_IF;
	
	IF #Weight_But = TRUE
	THEN
	    #Weight_DB := #Weight-#Weight_zero;
	    #P_w := #P;
	    #Weight_But := FALSE;
	END_IF;
	
	IF #Korect = TRUE
	THEN
	    #Weight_DB := (#S * (((#P_w - #P_z) / (9.81 * #Den)) * 100)) * #Den;
	    #Korect := FALSE;
	END_IF;
END_FUNCTION

FUNCTION_BLOCK "FB_Tank_Logic"
TITLE = Tank Coordinator
{ S7_Optimized_Access := 'FALSE' }
AUTHOR : Gemini
FAMILY : Archive
VERSION : 1.2
   VAR_INPUT 
      i_iRaw_AI { ExternalAccessible := 'False'; ExternalVisible := 'False'; ExternalWritable := 'False'} : Int;   // Аналоговый вход (PIW)
      i_rRaw_Siwa { ExternalAccessible := 'False'; ExternalVisible := 'False'; ExternalWritable := 'False'} : Real;   // Вес напрямую с Siwarex
      i_boRaw_DI { ExternalAccessible := 'False'; ExternalVisible := 'False'; ExternalWritable := 'False'} : Bool;   // Дискретный датчик (ВУ)
   END_VAR

   VAR_IN_OUT 
      io_Tank : "UDT_Tank_Full";   // Твои блоки как мультиэкземпляры
   END_VAR

   VAR 
      stat_AI { ExternalAccessible := 'False'; ExternalVisible := 'False'; ExternalWritable := 'False'} : "FB_AI";
      stat_AI_Alarm { ExternalAccessible := 'False'; ExternalVisible := 'False'; ExternalWritable := 'False'} : "FB_AI_Alarm";
      stat_DI { ExternalAccessible := 'False'; ExternalVisible := 'False'; ExternalWritable := 'False'} : "FB_DI";
      stat_DI_Alarm { ExternalAccessible := 'False'; ExternalVisible := 'False'; ExternalWritable := 'False'} : "FB_DI_Alarm";
   END_VAR

   VAR_TEMP 
      temp_Tank : "UDT_Tank_Full";
      temp_boIsSiwa : Bool;
      temp_boInhibitAI : Bool;
      temp_ResetError : Bool;
      temp_Value : Real;
   END_VAR


BEGIN
	// Ограничение компилятора S7-300/400:
	//      невозможно динамически пересчитать POINTER для вложенной IN_OUT структуры, потому используем временную переменную
	#temp_Tank := #io_Tank;
	
	// 0. ПРОВЕРКА НАЛИЧИЯ (Is_Present)
	// Если датчик не установлен в конфиге - не мучаем контроллер расчетами (DI_Conf.Mode = 3 канал отключен, AI_Conf.Mode - первый бит канал отключен)
	IF #temp_Tank.DI_Conf.Mode = "DB_Global".c_stDI_Mode.Disabled AND #temp_Tank.AI_Conf.Mode.Disabled THEN
	    RETURN;
	END_IF;
	
	// Читаем зафиксированную команду из слепка
	#temp_ResetError := #temp_Tank.Cmd.ResetError;
	// Если команда пришла, гасим ее НАПРЯМУЮ в io_Tank
	IF #temp_ResetError THEN
	    #io_Tank.Cmd.ResetError := FALSE;
	END_IF;
	
	// 1. ОБРАБОТКА АНАЛОГОВОГО КАНАЛА
	
	#stat_AI(i_iRawSignal := #i_iRaw_AI,
	         io_stConfig := #temp_Tank.AI_Conf,
	         io_stOut := #temp_Tank.AI_Out,
	         i_rSimValue := #i_rRaw_Siwa);
	
	
	// 2. ВЫЗОВ МАТЕМАТИКИ
	#temp_boIsSiwa := #temp_Tank.AI_Conf.Mode.SimActive;
	
	"FC_Tank_Calc"(i_rValue := #temp_Tank.AI_Out.Value_Filtered,
	               i_boIsSiwa := #temp_boIsSiwa,
	               io_Geom := #temp_Tank.Geom,
	               iq_Calc := #temp_Tank.Calc);
	
	// 3. АВАРИИ ПО УРОВНЮ (AI)
	// Глушим алармы AI при аппаратных ошибках (Inhibit)
	#temp_boInhibitAI := #temp_Tank.AI_Out.Status.WireBreak OR
	#temp_Tank.AI_Out.Status.Overflow OR
	#temp_Tank.AI_Out.Status.ConfigError;
	
	//В алармах обрабатываем реальный уровень, а не уровень без учета плотности(12 * 1.35 - датчик), или вес для весовых танков 
	IF #temp_boIsSiwa THEN
	    #temp_Value := #temp_Tank.Calc.Weight_t * 1000.0;// kg vs t ???
	ELSE
	    #temp_Value := #temp_Tank.Calc.Level_m;
	END_IF;
	
	#stat_AI_Alarm(i_rValue := #temp_Value, //#temp_Tank.AI_Out.Value_Filtered
	               i_boReset := #temp_ResetError,
	               i_boInhibit := #temp_boInhibitAI,
	               io_stConfig := #temp_Tank.AI_Alarm_Conf,
	               io_stOut := #temp_Tank.AI_Alarm);
	
	
	// 4. ОБРАБОТКА ДАТЧИКА ВЕРХНЕГО УРОВНЯ (DI)
	// Чистим дребезг
	#stat_DI(i_boRaw := #i_boRaw_DI,
	         io_stConfig := #temp_Tank.DI_Conf,
	         io_stOut := #temp_Tank.DI_Out);
	
	// Логика аварии ВУ (независима от AI)
	#stat_DI_Alarm(i_boSignal := #temp_Tank.DI_Out.Value,
	               i_boReset := #temp_ResetError,
	               i_boInhibit := (#temp_Tank.DI_Conf.Mode = "DB_Global".c_stDI_Mode.Disabled),
	               io_stConfig := #temp_Tank.DI_Alarm_Conf,
	               io_stOut := #temp_Tank.DI_Alarm);
	
	//Передаем только то что реально изменилось в ПЛК
	#io_Tank.AI_Out := #temp_Tank.AI_Out;
	#io_Tank.AI_Alarm := #temp_Tank.AI_Alarm;
	
	#io_Tank.DI_Out := #temp_Tank.DI_Out;
	#io_Tank.DI_Alarm := #temp_Tank.DI_Alarm;
	
	#io_Tank.Calc := #temp_Tank.Calc;
	
	
	
END_FUNCTION_BLOCK

FUNCTION "FC_Calc_Whause" : Void
{ S7_Optimized_Access := 'FALSE' }
VERSION : 0.1
   VAR_TEMP 
      temp_i : Int;
   END_VAR


BEGIN
	// ==============================================================================
	// СКЛАД TRN (3 танка)
	// ==============================================================================
	
	"DB_MAP".HMI_Whouse_TRN.Total_Volume_m3 := 0.0;
	"DB_MAP".HMI_Whouse_TRN.Total_Weight_t := 0.0;
	"DB_MAP".HMI_Whouse_TRN.Total_Ullage_pct := 0.0;
	"DB_MAP".HMI_Whouse_TRN.Total_Ullage_m3 := 0.0;
	"DB_MAP".HMI_Whouse_TRN.Tanks_In_Alarm := 0;
	
	FOR #temp_i := 1 TO "c_Count_TRN" DO
	    "FC_Wh_Totals_Aggregation"(io_Tanks := "DB_Wh_TRN".Tank[#temp_i],
	                               io_Whouse := "DB_MAP".HMI_Whouse_TRN);
	END_FOR;
	
	IF ("DB_MAP".HMI_Whouse_TRN.Total_Volume_m3 + "DB_MAP".HMI_Whouse_TRN.Total_Ullage_m3) >= 0.001 THEN
	    "DB_MAP".HMI_Whouse_TRN.Total_Ullage_pct :=
	    "DB_MAP".HMI_Whouse_TRN.Total_Ullage_m3 / ("DB_MAP".HMI_Whouse_TRN.Total_Volume_m3 + "DB_MAP".HMI_Whouse_TRN.Total_Ullage_m3) * 100.0;
	END_IF;
	
	"DB_MAP".HMI_Whouse_TRN.Status_Word.Global_Alarm := ("DB_MAP".HMI_Whouse_TRN.Tanks_In_Alarm > 0);
	
	// Сброс глобальной кнопки после прохода цикла
	IF "DB_MAP".HMI_Whouse_TRN.Cmd_Word.Reset_All THEN
	    "DB_MAP".HMI_Whouse_TRN.Cmd_Word.Reset_All := FALSE;
	END_IF;
	
	// ==============================================================================
	// СКЛАД POL (10 танков)
	// ==============================================================================
	"DB_MAP".HMI_Whouse_POL.Total_Volume_m3 := 0.0;
	"DB_MAP".HMI_Whouse_POL.Total_Weight_t := 0.0;
	"DB_MAP".HMI_Whouse_POL.Total_Ullage_pct := 0.0;
	"DB_MAP".HMI_Whouse_POL.Total_Ullage_m3 := 0.0;
	"DB_MAP".HMI_Whouse_POL.Tanks_In_Alarm := 0;
	
	FOR #temp_i := 1 TO "c_Count_POL" DO
	    "FC_Wh_Totals_Aggregation"(io_Tanks := "DB_Wh_POL".Tank[#temp_i],
	                               io_Whouse := "DB_MAP".HMI_Whouse_POL);
	END_FOR;
	
	IF ("DB_MAP".HMI_Whouse_POL.Total_Volume_m3 + "DB_MAP".HMI_Whouse_POL.Total_Ullage_m3) >= 0.001 THEN
	    "DB_MAP".HMI_Whouse_POL.Total_Ullage_pct :=
	    "DB_MAP".HMI_Whouse_POL.Total_Ullage_m3 / ("DB_MAP".HMI_Whouse_POL.Total_Volume_m3 + "DB_MAP".HMI_Whouse_POL.Total_Ullage_m3) * 100.0;
	END_IF;
	"DB_MAP".HMI_Whouse_POL.Status_Word.Global_Alarm := ("DB_MAP".HMI_Whouse_POL.Tanks_In_Alarm > 0);
	
	// Сброс глобальной кнопки после прохода цикла
	IF "DB_MAP".HMI_Whouse_POL.Cmd_Word.Reset_All THEN
	    "DB_MAP".HMI_Whouse_POL.Cmd_Word.Reset_All := FALSE;
	END_IF;
	
	// ==============================================================================
	// СКЛАД BUL (4 танка)
	// ==============================================================================
	"DB_MAP".HMI_Whouse_BUL.Total_Volume_m3 := 0.0;
	"DB_MAP".HMI_Whouse_BUL.Total_Weight_t := 0.0;
	"DB_MAP".HMI_Whouse_BUL.Total_Ullage_pct := 0.0;
	"DB_MAP".HMI_Whouse_BUL.Total_Ullage_m3 := 0.0;
	"DB_MAP".HMI_Whouse_BUL.Tanks_In_Alarm := 0;
	
	FOR #temp_i := 1 TO "c_Count_BUL" DO
	    "FC_Wh_Totals_Aggregation"(io_Tanks := "DB_Wh_BUL".Tank[#temp_i],
	                               io_Whouse := "DB_MAP".HMI_Whouse_BUL);
	END_FOR;
	
	IF ("DB_MAP".HMI_Whouse_BUL.Total_Volume_m3 + "DB_MAP".HMI_Whouse_BUL.Total_Ullage_m3) >= 0.001 THEN
	    "DB_MAP".HMI_Whouse_BUL.Total_Ullage_pct :=
	    "DB_MAP".HMI_Whouse_BUL.Total_Ullage_m3 / ("DB_MAP".HMI_Whouse_BUL.Total_Volume_m3 + "DB_MAP".HMI_Whouse_BUL.Total_Ullage_m3) * 100.0;
	END_IF;
	
	"DB_MAP".HMI_Whouse_BUL.Status_Word.Global_Alarm := ("DB_MAP".HMI_Whouse_BUL.Tanks_In_Alarm > 0);
	
	// Сброс глобальной кнопки после прохода цикла
	IF "DB_MAP".HMI_Whouse_BUL.Cmd_Word.Reset_All THEN
	    "DB_MAP".HMI_Whouse_BUL.Cmd_Word.Reset_All := FALSE;
	END_IF;
	
	// ==============================================================================
	// СКЛАД MOL (12 танков)
	// ==============================================================================
	"DB_MAP".HMI_Whouse_MOL.Total_Volume_m3 := 0.0;
	"DB_MAP".HMI_Whouse_MOL.Total_Weight_t := 0.0;
	"DB_MAP".HMI_Whouse_MOL.Total_Ullage_pct := 0.0;
	"DB_MAP".HMI_Whouse_MOL.Total_Ullage_m3 := 0.0;
	"DB_MAP".HMI_Whouse_MOL.Tanks_In_Alarm := 0;
	
	FOR #temp_i := 1 TO "c_Count_MOL" DO
	    "FC_Wh_Totals_Aggregation"(io_Tanks := "DB_Wh_MOL".Tank[#temp_i],
	                               io_Whouse := "DB_MAP".HMI_Whouse_MOL);
	END_FOR;
	
	IF ("DB_MAP".HMI_Whouse_MOL.Total_Volume_m3 + "DB_MAP".HMI_Whouse_MOL.Total_Ullage_m3) >= 0.001 THEN
	    "DB_MAP".HMI_Whouse_MOL.Total_Ullage_pct :=
	    "DB_MAP".HMI_Whouse_MOL.Total_Ullage_m3 / ("DB_MAP".HMI_Whouse_MOL.Total_Volume_m3 + "DB_MAP".HMI_Whouse_MOL.Total_Ullage_m3) * 100.0;
	END_IF;
	
	"DB_MAP".HMI_Whouse_MOL.Status_Word.Global_Alarm := ("DB_MAP".HMI_Whouse_MOL.Tanks_In_Alarm > 0);
	
	// Сброс глобальной кнопки после прохода цикла
	IF "DB_MAP".HMI_Whouse_MOL.Cmd_Word.Reset_All THEN
	    "DB_MAP".HMI_Whouse_MOL.Cmd_Word.Reset_All := FALSE;
	END_IF;
	
	
END_FUNCTION

FUNCTION "FC_Wh_Totals_Aggregation" : Void
{ S7_Optimized_Access := 'FALSE' }
VERSION : 0.1
   VAR_IN_OUT 
      io_Tanks : "UDT_Tank_Full";
      io_Whouse : "UDT_HMI_Whouse";
   END_VAR

   VAR_TEMP 
      temp_AnyAlarm : Bool;
   END_VAR


BEGIN
	        // Агрегация объемов и весов
	        #io_Whouse.Total_Volume_m3 := #io_Whouse.Total_Volume_m3 + #io_Tanks.Calc.Volume_m3;
	        #io_Whouse.Total_Weight_t := #io_Whouse.Total_Weight_t + #io_Tanks.Calc.Weight_t;
	        #io_Whouse.Total_Ullage_m3 := #io_Whouse.Total_Ullage_m3 + (#io_Tanks.Calc.Max_Volume_m3 - #io_Tanks.Calc.Volume_m3);
	        
	        // Проверка наличия аварий в танке (HH, H, L, LL или DI) 
	        IF #io_Tanks.AI_Alarm.HiHi OR
	            #io_Tanks.AI_Alarm.Hi OR
	            #io_Tanks.AI_Alarm.Lo OR
	            #io_Tanks.AI_Alarm.LoLo OR
	            #io_Tanks.DI_Alarm.Alarm
	        THEN
	            #io_Whouse.Tanks_In_Alarm := #io_Whouse.Tanks_In_Alarm + 1;
	        END_IF;
	        
	        // Трансляция глобальной команды "Сброс всех аварий" [cite: 56, 82]
	        IF #io_Whouse.Cmd_Reset_All THEN
	            #io_Tanks.Cmd.ResetError := TRUE;
	        END_IF;
END_FUNCTION

FUNCTION "FC_Log_Mng" : Void
{ S7_Optimized_Access := 'FALSE' }
VERSION : 0.1
   VAR_TEMP 
      temp_Ind : Int;
   END_VAR


BEGIN
	
	
	FOR #temp_Ind := 1 TO "c_Count_TRN" DO
	    "FC_Log_Tank"(i_Whouse_ID:=1,
	                  i_Tank_Index:=INT_TO_BYTE(#temp_Ind),
	              io_Tank:="DB_HMI_MAP".TRN_SmalTank[#temp_Ind]);
	END_FOR;
	
	FOR #temp_Ind := 1 TO "c_Count_POL" DO
	    "FC_Log_Tank"(i_Whouse_ID := 2,
	                  i_Tank_Index := INT_TO_BYTE(#temp_Ind),
	                  io_Tank := "DB_HMI_MAP".POL_SmalTank[#temp_Ind]);
	END_FOR;
	
	FOR #temp_Ind := 1 TO "c_Count_BUL" DO
	    "FC_Log_Tank"(i_Whouse_ID := 3,
	                  i_Tank_Index := INT_TO_BYTE(#temp_Ind),
	                  io_Tank := "DB_HMI_MAP".BUL_SmalTank[#temp_Ind]);
	END_FOR;
	
	FOR #temp_Ind := 1 TO "c_Count_MOL" DO
	    "FC_Log_Tank"(i_Whouse_ID := 4,
	                  i_Tank_Index := INT_TO_BYTE(#temp_Ind),
	                  io_Tank := "DB_HMI_MAP".MOL_SmalTank[#temp_Ind]);
	END_FOR;
	
END_FUNCTION

FUNCTION "FC_Log_Tank" : Void
{ S7_Optimized_Access := 'FALSE' }
VERSION : 0.1
   VAR_INPUT 
      i_Whouse_ID : Byte;
      i_Tank_Index : Byte;
   END_VAR

   VAR_IN_OUT 
      io_Tank : "UDT_HMI_SmallTank";
   END_VAR

   VAR_TEMP 
      temp_Write_Ptr : Int;
      temp_DT : Date_And_Time;
   END_VAR


BEGIN
	
	#temp_DT := "DB_DateTime".DateTime_PLC;
	#temp_Write_Ptr := "DB_Log_Buffer".Write_Index;
	
	"DB_Log_Buffer".Buffer[#temp_Write_Ptr].Timestamp := #temp_DT;
	"DB_Log_Buffer".Buffer[#temp_Write_Ptr].Whouse_ID := #i_Whouse_ID;
	"DB_Log_Buffer".Buffer[#temp_Write_Ptr].Tank_Index := #i_Tank_Index;
	"DB_Log_Buffer".Buffer[#temp_Write_Ptr].Level_m := #io_Tank.Level_m;
	"DB_Log_Buffer".Buffer[#temp_Write_Ptr].Weight_t := #io_Tank.Weight_t;
	//"DB_Log_Buffer".Buffer[#temp_Write_Ptr].Status_Bits := #temp_Status;
	
	#temp_Write_Ptr := #temp_Write_Ptr + 1;
	IF #temp_Write_Ptr > 1999 THEN
	    #temp_Write_Ptr := 0;
	END_IF;
END_FUNCTION

FUNCTION "FC_Wh_BUL_Mng" : Void
{ S7_Optimized_Access := 'FALSE' }
VERSION : 0.1
   VAR_TEMP 
      temp_Ind : Int;
   END_VAR


BEGIN
	// ---------------------------------------------------------------
	// Склад: Болгарский (BUL) — 4 танка
	// ---------------------------------------------------------------
	
	"iDB_BUL_Tank_Log_1"(i_iRaw_AI := "DB_IO_MAP".AI_BUL_Tank_1,
	                     i_rRaw_Siwa := 0.0,
	                     i_boRaw_DI := "DB_IO_MAP".DI_BUL_Tank_1,
	                     io_Tank := "DB_Wh_BUL".Tank[1]);
	
	"iDB_BUL_Tank_Log_2"(i_iRaw_AI := "DB_IO_MAP".AI_BUL_Tank_2,
	                     i_rRaw_Siwa := 0.0,
	                     i_boRaw_DI := "DB_IO_MAP".DI_BUL_Tank_2,
	                     io_Tank := "DB_Wh_BUL".Tank[2]);
	
	"iDB_BUL_Tank_Log_3"(i_iRaw_AI := "DB_IO_MAP".AI_BUL_Tank_3,
	                     i_rRaw_Siwa := 0.0,
	                     i_boRaw_DI := "DB_IO_MAP".DI_BUL_Tank_3,
	                     io_Tank := "DB_Wh_BUL".Tank[3]);
	
	"iDB_BUL_Tank_Log_4"(i_iRaw_AI := "DB_IO_MAP".AI_BUL_Tank_4,
	                     i_rRaw_Siwa := 0.0,
	                     i_boRaw_DI := "DB_IO_MAP".DI_BUL_Tank_4,
	                     io_Tank := "DB_Wh_BUL".Tank[4]);
	
	// HMI маппинг
	FOR #temp_Ind := 1 TO "c_Count_BUL" DO
	    "FC_Map_SmallTank_HMI"(io_Tank_Internal := "DB_Wh_BUL".Tank[#temp_Ind],
	                           io_HMI_Tank := "DB_HMI_MAP".BUL_SmalTank[#temp_Ind]);
	END_FOR;
	
END_FUNCTION

FUNCTION "FC_Wh_MOL_Mng" : Void
{ S7_Optimized_Access := 'FALSE' }
VERSION : 0.1
   VAR_TEMP 
      temp_Ind : Int;
   END_VAR


BEGIN
	// ---------------------------------------------------------------
	// Склад: Молдавский (MOL) — 12 танков
	// ---------------------------------------------------------------
	
	"iDB_MOL_Tank_Log_1"(i_iRaw_AI := "DB_IO_MAP".AI_MOL_Tank_1,
	                     i_rRaw_Siwa := 0.0,
	                     i_boRaw_DI := "DB_IO_MAP".DI_MOL_Tank_1,
	                     io_Tank := "DB_Wh_MOL".Tank[1]);
	
	"iDB_MOL_Tank_Log_2"(i_iRaw_AI := "DB_IO_MAP".AI_MOL_Tank_2,
	                     i_rRaw_Siwa := 0.0,
	                     i_boRaw_DI := "DB_IO_MAP".DI_MOL_Tank_2,
	                     io_Tank := "DB_Wh_MOL".Tank[2]);
	
	"iDB_MOL_Tank_Log_3"(i_iRaw_AI := "DB_IO_MAP".AI_MOL_Tank_3,
	                     i_rRaw_Siwa := 0.0,
	                     i_boRaw_DI := "DB_IO_MAP".DI_MOL_Tank_3,
	                     io_Tank := "DB_Wh_MOL".Tank[3]);
	
	"iDB_MOL_Tank_Log_4"(i_iRaw_AI := "DB_IO_MAP".AI_MOL_Tank_4,
	                     i_rRaw_Siwa := 0.0,
	                     i_boRaw_DI := "DB_IO_MAP".DI_MOL_Tank_4,
	                     io_Tank := "DB_Wh_MOL".Tank[4]);
	
	"iDB_MOL_Tank_Log_5"(i_iRaw_AI := "DB_IO_MAP".AI_MOL_Tank_5,
	                     i_rRaw_Siwa := 0.0,
	                     i_boRaw_DI := "DB_IO_MAP".DI_MOL_Tank_5,
	                     io_Tank := "DB_Wh_MOL".Tank[5]);
	
	"iDB_MOL_Tank_Log_6"(i_iRaw_AI := "DB_IO_MAP".AI_MOL_Tank_6,
	                     i_rRaw_Siwa := 0.0,
	                     i_boRaw_DI := "DB_IO_MAP".DI_MOL_Tank_6,
	                     io_Tank := "DB_Wh_MOL".Tank[6]);
	
	"iDB_MOL_Tank_Log_7"(i_iRaw_AI := "DB_IO_MAP".AI_MOL_Tank_7,
	                     i_rRaw_Siwa := 0.0,
	                     i_boRaw_DI := "DB_IO_MAP".DI_MOL_Tank_7,
	                     io_Tank := "DB_Wh_MOL".Tank[7]);
	
	"iDB_MOL_Tank_Log_8"(i_iRaw_AI := "DB_IO_MAP".AI_MOL_Tank_8,
	                     i_rRaw_Siwa := 0.0,
	                     i_boRaw_DI := "DB_IO_MAP".DI_MOL_Tank_8,
	                     io_Tank := "DB_Wh_MOL".Tank[8]);
	
	"iDB_MOL_Tank_Log_9"(i_iRaw_AI := "DB_IO_MAP".AI_MOL_Tank_9,
	                     i_rRaw_Siwa := 0.0,
	                     i_boRaw_DI := "DB_IO_MAP".DI_MOL_Tank_9,
	                     io_Tank := "DB_Wh_MOL".Tank[9]);
	
	"iDB_MOL_Tank_Log_10"(i_iRaw_AI := "DB_IO_MAP".AI_MOL_Tank_10,
	                      i_rRaw_Siwa := 0.0,
	                      i_boRaw_DI := "DB_IO_MAP".DI_MOL_Tank_10,
	                      io_Tank := "DB_Wh_MOL".Tank[10]);
	
	"iDB_MOL_Tank_Log_11"(i_iRaw_AI := "DB_IO_MAP".AI_MOL_Tank_11,
	                      i_rRaw_Siwa := 0.0,
	                      i_boRaw_DI := "DB_IO_MAP".DI_MOL_Tank_11,
	                      io_Tank := "DB_Wh_MOL".Tank[11]);
	
	"iDB_MOL_Tank_Log_12"(i_iRaw_AI := "DB_IO_MAP".AI_MOL_Tank_12,
	                      i_rRaw_Siwa := 0.0,
	                      i_boRaw_DI := "DB_IO_MAP".DI_MOL_Tank_12,
	                      io_Tank := "DB_Wh_MOL".Tank[12]);
	
	// HMI маппинг
	FOR #temp_Ind := 1 TO "c_Count_MOL" DO
	    "FC_Map_SmallTank_HMI"(io_Tank_Internal := "DB_Wh_MOL".Tank[#temp_Ind],
	                           io_HMI_Tank := "DB_HMI_MAP".MOL_SmalTank[#temp_Ind]);
	END_FOR;
END_FUNCTION

FUNCTION_BLOCK "CalculationVolume"
{ S7_Optimized_Access := 'FALSE' }
VERSION : 0.1
   VAR_INPUT 
      IW_Radius : Real;
      IW_ValueFromSensor : Real;
      IW_K_for_Tonnag : Real;
      IW_K_for_Level : Real;
   END_VAR

   VAR_OUTPUT 
      QW_Volume : Real;
      QW_Tonnag : Real;
      QW_RealLevel : Real;
   END_VAR

   VAR 
      sW_S : Real;
      sW_Volume : Real;
      sW_RealLevel : Real;
   END_VAR

   VAR CONSTANT 
      const_PI : Real := 3.14;
   END_VAR


BEGIN
	// Обрахування реального рівня
	#sW_RealLevel := #IW_ValueFromSensor / #IW_K_for_Level;
	
	// Обрахування площа перерізу 1 - для ємності,
	#sW_S := #const_PI * #IW_Radius * #IW_Radius;
	    
	// Volume = об*єм
	#sW_Volume := #sW_S * #sW_RealLevel;
	
	#QW_RealLevel := #sW_RealLevel; //реальний рівень
	#QW_Volume := #sW_Volume; //Присвоєння обрахованого обєму на вихід
	#QW_Tonnag := #sW_Volume * #IW_K_for_Tonnag; // обрахований обєм * Коефіцієнт
END_FUNCTION_BLOCK

FUNCTION "LevelTanks" : Void
{ S7_Optimized_Access := 'FALSE' }
VERSION : 0.1

BEGIN
	
	REGION Polska - Tank 1
	    
	    "AI_Tank1_DB"(IB_Reset_PLC := "Total_DB".Restart_PLC,
	                  IB_Total_Reset := "Total_DB".Total_Reset_HMI,
	                  IB_EnablePowerControl := FALSE,
	                  IW_HW_UpLevel := 27648,
	                  IW_HW_LowLevel := 0,
	                  IW_Signal_from_Sensor := "IW_Tank1",
	                  IUDT_Analog_In := "UDT_AI_Tank1");
	    
	 "CalcVolume_Tank1_DB"(IW_ValueFromSensor:="AI_Tank1_DB".QDW_ScalledValue);
	 
	END_REGION
	
	REGION Polska - Tank 2
	    
	    "AI_Tank2_DB"(IB_Reset_PLC := "Total_DB".Restart_PLC,
	                  IB_Total_Reset := "Total_DB".Total_Reset_HMI,
	                  IB_EnablePowerControl := FALSE,
	                  IW_HW_UpLevel := 27648,
	                  IW_HW_LowLevel := 0,
	                  IW_Signal_from_Sensor := "IW_Tank2",
	                  IUDT_Analog_In := "UDT_AI_Tank2");
	    
	    "CalcVolume_Tank2_DB"(IW_ValueFromSensor := "AI_Tank2_DB".QDW_ScalledValue);
	    
	END_REGION
	
	REGION Polska - Tank 3
	    
	    "AI_Tank3_DB"(IB_Reset_PLC := "Total_DB".Restart_PLC,
	                  IB_Total_Reset := "Total_DB".Total_Reset_HMI,
	                  IB_EnablePowerControl := FALSE,
	                  IW_HW_UpLevel := 27648,
	                  IW_HW_LowLevel := 0,
	                  IW_Signal_from_Sensor := "IW_Tank3",
	                  IUDT_Analog_In := "UDT_AI_Tank3");
	    
	    "CalcVolume_Tank3_DB"(IW_ValueFromSensor := "AI_Tank3_DB".QDW_ScalledValue);
	    
	END_REGION
	
	REGION Polska - Tank 4
	    
	    "AI_Tank4_DB"(IB_Reset_PLC := "Total_DB".Restart_PLC,
	                  IB_Total_Reset := "Total_DB".Total_Reset_HMI,
	                  IB_EnablePowerControl := FALSE,
	                  IW_HW_UpLevel := 27648,
	                  IW_HW_LowLevel := 0,
	                  IW_Signal_from_Sensor := "IW_Tank4",
	                  IUDT_Analog_In := "UDT_AI_Tank4");
	    
	    "CalcVolume_Tank4_DB"(IW_ValueFromSensor := "AI_Tank4_DB".QDW_ScalledValue);
	    
	END_REGION
	
	REGION Polska - Tank 5
	    
	    "AI_Tank5_DB"(IB_Reset_PLC := "Total_DB".Restart_PLC,
	                  IB_Total_Reset := "Total_DB".Total_Reset_HMI,
	                  IB_EnablePowerControl := FALSE,
	                  IW_HW_UpLevel := 27648,
	                  IW_HW_LowLevel := 0,
	                  IW_Signal_from_Sensor := "IW_Tank5",
	                  IUDT_Analog_In := "UDT_AI_Tank5");
	    
	    "CalcVolume_Tank5_DB"(IW_ValueFromSensor := "AI_Tank5_DB".QDW_ScalledValue);
	    
	END_REGION
	
	REGION Polska - Tank 6
	    
	    "AI_Tank6_DB"(IB_Reset_PLC := "Total_DB".Restart_PLC,
	                  IB_Total_Reset := "Total_DB".Total_Reset_HMI,
	                  IB_EnablePowerControl := FALSE,
	                  IW_HW_UpLevel := 27648,
	                  IW_HW_LowLevel := 0,
	                  IW_Signal_from_Sensor := "IW_Tank6",
	                  IUDT_Analog_In := "UDT_AI_Tank6");
	    
	    "CalcVolume_Tank6_DB"(IW_ValueFromSensor := "AI_Tank6_DB".QDW_ScalledValue);
	    
	END_REGION
	
	REGION Polska - Tank 7
	    
	    "AI_Tank7_DB"(IB_Reset_PLC := "Total_DB".Restart_PLC,
	                  IB_Total_Reset := "Total_DB".Total_Reset_HMI,
	                  IB_EnablePowerControl := FALSE,
	                  IW_HW_UpLevel := 27648,
	                  IW_HW_LowLevel := 0,
	                  IW_Signal_from_Sensor := "IW_Tank7",
	                  IUDT_Analog_In := "UDT_AI_Tank7");
	    
	    "CalcVolume_Tank7_DB"(IW_ValueFromSensor := "AI_Tank7_DB".QDW_ScalledValue);
	    
	END_REGION
	
	REGION Polska - Tank 8
	    
	    "AI_Tank8_DB"(IB_Reset_PLC := "Total_DB".Restart_PLC,
	                  IB_Total_Reset := "Total_DB".Total_Reset_HMI,
	                  IB_EnablePowerControl := FALSE,
	                  IW_HW_UpLevel := 27648,
	                  IW_HW_LowLevel := 0,
	                  IW_Signal_from_Sensor := "IW_Tank8",
	                  IUDT_Analog_In := "UDT_AI_Tank8");
	    
	    "CalcVolume_Tank8_DB"(IW_ValueFromSensor := "AI_Tank8_DB".QDW_ScalledValue);
	    
	END_REGION
	
	REGION Polska - Tank 9
	    
	    "AI_Tank9_DB"(IB_Reset_PLC := "Total_DB".Restart_PLC,
	                  IB_Total_Reset := "Total_DB".Total_Reset_HMI,
	                  IB_EnablePowerControl := FALSE,
	                  IW_HW_UpLevel := 27648,
	                  IW_HW_LowLevel := 0,
	                  IW_Signal_from_Sensor := "IW_Tank9",
	                  IUDT_Analog_In := "UDT_AI_Tank9");
	    
	    "CalcVolume_Tank9_DB"(IW_ValueFromSensor := "AI_Tank9_DB".QDW_ScalledValue);
	    
	END_REGION
	
	REGION Polska - Tank 10
	    
	    "AI_Tank10_DB"(IB_Reset_PLC := "Total_DB".Restart_PLC,
	                  IB_Total_Reset := "Total_DB".Total_Reset_HMI,
	                  IB_EnablePowerControl := FALSE,
	                  IW_HW_UpLevel := 27648,
	                  IW_HW_LowLevel := 0,
	                  IW_Signal_from_Sensor := "IW_Tank10",
	                  IUDT_Analog_In := "UDT_AI_Tank10");
	    
	    "CalcVolume_Tank10_DB"(IW_ValueFromSensor := "AI_Tank10_DB".QDW_ScalledValue);
	    
	END_REGION
	
	REGION Bolgarska - Tank 1
	    
	    "AI_Tank11_DB"(IB_Reset_PLC := "Total_DB".Restart_PLC,
	                  IB_Total_Reset := "Total_DB".Total_Reset_HMI,
	                  IB_EnablePowerControl := FALSE,
	                  IW_HW_UpLevel := 27648,
	                  IW_HW_LowLevel := 0,
	                  IW_Signal_from_Sensor := "IW_Tank11",
	                  IUDT_Analog_In := "UDT_AI_Tank11");
	    
	    "CalcVolume_Tank11_DB"(IW_ValueFromSensor := "AI_Tank11_DB".QDW_ScalledValue);
	    
	END_REGION
	
	REGION Bolgarska - Tank 2
	    
	    "AI_Tank12_DB"(IB_Reset_PLC := "Total_DB".Restart_PLC,
	                  IB_Total_Reset := "Total_DB".Total_Reset_HMI,
	                  IB_EnablePowerControl := FALSE,
	                  IW_HW_UpLevel := 27648,
	                  IW_HW_LowLevel := 0,
	                  IW_Signal_from_Sensor := "IW_Tank12",
	                  IUDT_Analog_In := "UDT_AI_Tank12");
	    
	    "CalcVolume_Tank12_DB"(IW_ValueFromSensor := "AI_Tank12_DB".QDW_ScalledValue);
	    
	END_REGION
	
	REGION Bolgarska - Tank 3
	    
	    "AI_Tank13_DB"(IB_Reset_PLC := "Total_DB".Restart_PLC,
	                   IB_Total_Reset := "Total_DB".Total_Reset_HMI,
	                   IB_EnablePowerControl := FALSE,
	                   IW_HW_UpLevel := 27648,
	                   IW_HW_LowLevel := 0,
	                   IW_Signal_from_Sensor := "IW_Tank13", // Задати 
	                   IUDT_Analog_In := "UDT_AI_Tank13");
	    
	    "CalcVolume_Tank13_DB"(IW_ValueFromSensor := "AI_Tank13_DB".QDW_ScalledValue);
	    
	END_REGION
	
	REGION Bolgarska - Tank 4
	    
	    "AI_Tank14_DB"(IB_Reset_PLC := "Total_DB".Restart_PLC,
	                   IB_Total_Reset := "Total_DB".Total_Reset_HMI,
	                   IB_EnablePowerControl := FALSE,
	                   IW_HW_UpLevel := 27648,
	                   IW_HW_LowLevel := 0,
	                   IW_Signal_from_Sensor := "IW_Tank14", // Задати 
	                   IUDT_Analog_In := "UDT_AI_Tank14");
	    
	    "CalcVolume_Tank14_DB"(IW_ValueFromSensor := "AI_Tank14_DB".QDW_ScalledValue);
	    
	END_REGION
	
	
	
END_FUNCTION

FUNCTION_BLOCK "Analog_In_UDT"
{ S7_Optimized_Access := 'FALSE' }
AUTHOR : SimenCom
VERSION : 1.0
   VAR_INPUT 
      IB_Reset_PLC : Bool := false;
      IB_Total_Reset : Bool := false;
      IB_EnablePowerControl : Bool;
      IB_PowerControl : Bool;
      IW_HW_UpLevel : Int;
      IW_HW_LowLevel : Int;
      IW_Signal_from_Sensor : Int := 0;
   END_VAR

   VAR_OUTPUT 
      QW_STW : Array[0..15] of Bool;
      QDW_ScalledValue : Real;
      QB_HiHi_Fault : Bool;
      QB_Hi_Alarm : Bool;
      QB_Lo_Alarm : Bool;
      QB_LoLo_Fault : Bool;
      QB_Sensor_in_Zero : Bool;
   END_VAR

   VAR_IN_OUT 
      IUDT_Analog_In : "UDT_Analog_In";
   END_VAR

   VAR 
      Timer_TON_Filter {InstructionName := 'TON'; LibVersion := '1.0'} : TON;
      StB_Filter { ExternalAccessible := 'False'; ExternalVisible := 'False'; ExternalWritable := 'False'} : Bool;
      StDW_Sensor_After_Filter { ExternalAccessible := 'False'; ExternalVisible := 'False'; ExternalWritable := 'False'} : Real;
      StDW_Sensor_After_Scaling : Real;
      StB_HiHi : Bool;
      StB_Hi : Bool;
      StB_LoLo : Bool;
      StB_Lo : Bool;
      StB_HiHi_Q : Bool;
      StB_Hi_Q : Bool;
      StB_LoLo_Q : Bool;
      StB_Lo_Q : Bool;
      StB_PowerFault : Bool;
      Level_Control_HoLo : "Level_Control_HoLo";
      Smoothing_Instance : "Smoothing";
      Level_Control_HoLo_Instance : "Level_Control_HoLo";
   END_VAR

   VAR_TEMP 
      TmDW_Sensor_in_real : Real;
      TmB_Fault : Bool;
      TmDW_Sensor_After_DeadZone : Real;
      TmB_Reset_Bit : Bool;
      TmB_Sensor_In_Zero : Bool;
      TmDW_OutVal : Real;
   END_VAR


BEGIN
	// Help info 
	(*Біти в контрольних
	    словах:
	IW_CTW              
	0   -   Скиданя помилки -Кнопка-    SetBit
	1   -   Ввімкнути симуляцію -"Галочка"- SetBit
	2   -           
	3   -           
	4   -           
	5   -           
	6   -           
	7   -           
	8   -           
	9   -           
	10  -           
	11  -           
	12  -           
	13  -           
	14  -           
	15  -           
	    ************************************************************************
	    ************************************************************************
	QLW_STW     
	0   -   Все добре
	1   -   Активне попередження
	2   -   Загальна аварія
	3   -   Сигнал обриву давача 
	4   -   Досягнуто аварійного рівня (HiHi)
	5   -   Досягнуто рівня попередження (Hi)
	6   -   Опустилося нижче рівня попередження (Lo)
	7   -   Опустилося нижче аварійного рівня (LoLo)
	8   -   Симуляція ввімкнена
	9   -   Активне скидання помилок
	10  -   
	11  -   
	12  -   
	13  -   
	14  -   
	15  -   
	
	    ************************************************************************
	    ************************************************************************
	QDW_Message              
	0   -   Обрив лінії давача  -   Аварія
	1   -   Досягнуто аварійного рівня (HiHi)   -   Аварія
	2   -   Опустилося нижче аварійного рівня (LoLo)    -   Аварія
	3   -       -   
	4   -       -   
	5   -       -   
	6   -       -   
	7   -       -   
	8   -       -   
	9   -       -   
	10  -           
	11  -           
	12  -       -   
	13  -       -   
	14  -   Досягнуто рівня попередження (Hi)   -   Попередження
	15  -   Опустилося нижче рівня попередження (Lo)    -   Попередження
	16  -   Симуляція ввімкнена -   Подія
	17  -       -   
	18  -       -   
	19  -       -   
	20  -       -   
	
	*) 
	//Reset
	#TmB_Reset_Bit := #IB_Reset_PLC OR #IB_Total_Reset OR #IUDT_Analog_In.IW_CTW[0];
	
	//Логіка елементі живлення давача
	IF #IB_EnablePowerControl THEN
	    // #F_TRIG_PowerControl(CLK := #IB_PowerControl);
	    #StB_PowerFault := NOT #IB_PowerControl OR (#StB_PowerFault AND NOT #TmB_Reset_Bit);
	ELSE
	    #StB_PowerFault := false;
	END_IF;
	
	
	
	
	//Обрив давача
	IF  #IW_Signal_from_Sensor <= -32768 OR #IW_Signal_from_Sensor >= 32767 OR ((#StB_PowerFault OR NOT #IB_PowerControl) AND #IB_EnablePowerControl)  THEN
	    #TmB_Sensor_In_Zero := True;
	    #QB_Sensor_in_Zero := True;
	ELSE
	    #TmB_Sensor_In_Zero := False;
	    #QB_Sensor_in_Zero := False;
	END_IF;
	
	#TmDW_Sensor_in_real := INT_TO_REAL(#IW_Signal_from_Sensor);
	#IUDT_Analog_In.QW_HWValue := #IW_Signal_from_Sensor;
	
	// Згладжування сигналу . Масивне згладжування. Максимум 60 секунд
	#Smoothing_Instance(IDW_Input_Value := #TmDW_Sensor_in_real,
	                    IW_Time_Smoothing := #IUDT_Analog_In.IW_Time_Filter,
	                    IB_Gen_In := "tag_1",
	                    IW_Gen_Value := 200,
	                    QDW_Smoothing_Value => #StDW_Sensor_After_Filter);
	
	#TmDW_Sensor_in_real := 0;
	
	//Масштабування сигналу з множенням на коофіцієнт
	"Scaling_TSS"(In_Value := #StDW_Sensor_After_Filter,
	              In_Max := #IW_HW_UpLevel,
	              In_Min := #IW_HW_LowLevel,
	              Out_Max := #IUDT_Analog_In.IDW_UpLevel,
	              Out_Min := #IUDT_Analog_In.IDW_LowLevel,
	              Out_Value => #TmDW_OutVal,
	              Fault => #TmB_Fault,
	              Senser_In_Zero => #TmB_Fault);
	#StDW_Sensor_After_Scaling := #TmDW_OutVal * #IUDT_Analog_In.IDW_K_Mult;
	// "Мертва зона" сенсора
	IF #StDW_Sensor_After_Scaling >= #IUDT_Analog_In.IDW_DeadZone THEN
	#TmDW_Sensor_After_DeadZone := #StDW_Sensor_After_Scaling;
	ELSE
	    #TmDW_Sensor_After_DeadZone := 0;
	END_IF;
	
	
	// Обмеження симуляційного завдання
	IF #IUDT_Analog_In.IDW_Simulation_Value > #IUDT_Analog_In.IDW_UpLevel * #IUDT_Analog_In.IDW_K_Mult  THEN
	    #IUDT_Analog_In.IDW_Simulation_Value := #IUDT_Analog_In.IDW_UpLevel * #IUDT_Analog_In.IDW_K_Mult ;
	ELSIF #IUDT_Analog_In.IDW_Simulation_Value < #IUDT_Analog_In.IDW_LowLevel * #IUDT_Analog_In.IDW_K_Mult THEN
	    #IUDT_Analog_In.IDW_Simulation_Value := #IUDT_Analog_In.IDW_LowLevel * #IUDT_Analog_In.IDW_K_Mult ;
	END_IF;
	#TmDW_Sensor_in_real := 0;
	
	// Симуляція
	IF #IUDT_Analog_In.IW_CTW[0] THEN
	    #TmDW_Sensor_in_real := #IUDT_Analog_In.IDW_Simulation_Value;
	    #IUDT_Analog_In.QW_STW[8] := True;
	    
	ELSE
	    #TmDW_Sensor_in_real := #TmDW_Sensor_After_DeadZone;
	    #IUDT_Analog_In.QW_STW[8] := False;
	END_IF;
	
	//Блокування виходу при обриві
	IF NOT #TmB_Sensor_In_Zero OR #IUDT_Analog_In.IW_CTW[1] THEN
	    #QDW_ScalledValue := #TmDW_Sensor_in_real;
	    #IUDT_Analog_In.QDW_ScalledValue := #TmDW_Sensor_in_real;
	ELSE
	    #QDW_ScalledValue := 0.0;
	    #IUDT_Analog_In.QDW_ScalledValue := 0.0;
	    #TmDW_Sensor_in_real := 0.0;
	END_IF;
	
	// Логіка орпцювання аварійних повідомлень по сенсору
	// #IUDT_Analog_In.IBt_Block_ControlLevel.%X0 := true;
	// #IUDT_Analog_In.IBt_Block_ControlLevel.%X1 := true;
	// #IUDT_Analog_In.IBt_Block_ControlLevel.%X2 := true;
	// #IUDT_Analog_In.IBt_Block_ControlLevel.%X3 := true;
	#Level_Control_HoLo(IB_Enable_Func := NOT #TmB_Sensor_In_Zero,
	                    IDW_Actual_Value := #TmDW_Sensor_in_real,
	                    IDW_Set_HiHi := #IUDT_Analog_In.IDW_HiHi,
	                    IDW_Set_Hi := #IUDT_Analog_In.IDW_Hi,
	                    IDW_Set_LoLo := #IUDT_Analog_In.IDW_Lolo,
	                    IDW_Set_Lo := #IUDT_Analog_In.IDW_Lo,
	                    IW_Time_HiHi := #IUDT_Analog_In.IW_DelayON_HiHi,
	                    IW_Time_Hi := #IUDT_Analog_In.IW_DelayON_Hi,
	                    IW_Time_LoLo := #IUDT_Analog_In.IW_DelayON_LoLo,
	                    IW_Time_Lo := #IUDT_Analog_In.IW_DelayON_Lo);
	#StB_HiHi := (#StB_HiHi AND NOT #TmB_Reset_Bit)
	OR #IUDT_Analog_In.IBt_Enable_ControlLevel[0] AND #Level_Control_HoLo.QB_HiHi;
	#StB_HiHi_Q := (#StB_HiHi_Q AND NOT #TmB_Reset_Bit)
	OR #Level_Control_HoLo.QB_HiHi AND #IUDT_Analog_In.IBt_Block_ControlLevel[0];
	#QB_HiHi_Fault := #StB_HiHi_Q;
	
